      movel([0.226633, -1.444868, -2.521019, -0.746502, 1.570796, 1.797429],accel_mss,speed_ms,0,blend_radius_m)
      movel([0.225647, -1.445273, -2.520694, -0.746422, 1.570796, 1.796443],accel_mss,speed_ms,0,blend_radius_m)
      movel([0.224501, -1.445732, -2.520325, -0.746331, 1.570796, 1.795298],accel_mss,speed_ms,0,blend_radius_m)
      movel([0.221549, -1.446906, -2.519382, -0.746101, 1.570796, 1.792346],accel_mss,speed_ms,0,blend_radius_m)
      movel([0.221114, -1.448639, -2.517985, -0.745765, 1.570796, 1.791910],accel_mss,speed_ms,0,blend_radius_m)
      movel([0.220680, -1.450369, -2.516586, -0.745434, 1.570796, 1.791476],accel_mss,speed_ms,0,blend_radius_m)
      movel([0.218279, -1.451481, -2.515684, -0.745224, 1.570796, 1.789076],accel_mss,speed_ms,0,blend_radius_m)
      movel([0.215883, -1.452595, -2.514779, -0.745015, 1.570796, 1.786679],accel_mss,speed_ms,0,blend_radius_m)
      movel([0.215624, -1.453437, -2.514093, -0.744859, 1.570796, 1.786421],accel_mss,speed_ms,0,blend_radius_m)
      movel([0.215367, -1.454275, -2.513410, -0.744704, 1.570796, 1.786163],accel_mss,speed_ms,0,blend_radius_m)
      movel([0.192396, -1.457892, -2.510448, -0.744049, 1.570796, 1.763193],accel_mss,speed_ms,0,blend_radius_m)
      movel([0.169430, -1.461921, -2.507125, -0.743343, 1.570796, 1.740226],accel_mss,speed_ms,0,blend_radius_m)
      movel([0.170007, -1.461323, -2.507620, -0.743446, 1.570796, 1.740803],accel_mss,speed_ms,0,blend_radius_m)
      movel([0.170664, -1.460630, -2.508192, -0.743566, 1.570796, 1.741460],accel_mss,speed_ms,0,blend_radius_m)
      movel([0.171304, -1.459927, -2.508773, -0.743689, 1.570796, 1.742101],accel_mss,speed_ms,0,blend_radius_m)
      movel([0.171930, -1.459214, -2.509360, -0.743814, 1.570796, 1.742727],accel_mss,speed_ms,0,blend_radius_m)
      movel([0.172537, -1.458492, -2.509955, -0.743942, 1.570796, 1.743334],accel_mss,speed_ms,0,blend_radius_m)
      movel([0.173093, -1.457802, -2.510522, -0.744065, 1.570796, 1.743889],accel_mss,speed_ms,0,blend_radius_m)
      movel([0.173629, -1.457105, -2.511094, -0.744190, 1.570796, 1.744425],accel_mss,speed_ms,0,blend_radius_m)
      movel([0.174144, -1.456397, -2.511674, -0.744317, 1.570796, 1.744940],accel_mss,speed_ms,0,blend_radius_m)
      movel([0.174639, -1.455683, -2.512259, -0.744447, 1.570796, 1.745435],accel_mss,speed_ms,0,blend_radius_m)
      movel([0.175094, -1.454986, -2.512830, -0.744574, 1.570796, 1.745891],accel_mss,speed_ms,0,blend_radius_m)
      movel([0.175530, -1.454281, -2.513405, -0.744703, 1.570796, 1.746326],accel_mss,speed_ms,0,blend_radius_m)
      movel([0.175941, -1.453573, -2.513982, -0.744834, 1.570796, 1.746737],accel_mss,speed_ms,0,blend_radius_m)
      movel([0.176327, -1.452859, -2.514564, -0.744966, 1.570796, 1.747124],accel_mss,speed_ms,0,blend_radius_m)
      movel([0.176693, -1.452141, -2.515148, -0.745100, 1.570796, 1.747489],accel_mss,speed_ms,0,blend_radius_m)
      movel([0.177031, -1.451421, -2.515732, -0.745235, 1.570796, 1.747828],accel_mss,speed_ms,0,blend_radius_m)
      movel([0.177346, -1.450701, -2.516317, -0.745371, 1.570796, 1.748142],accel_mss,speed_ms,0,blend_radius_m)
      movel([0.177636, -1.449977, -2.516903, -0.745509, 1.570796, 1.748432],accel_mss,speed_ms,0,blend_radius_m)
      movel([0.177833, -1.449428, -2.517348, -0.745614, 1.570796, 1.748629],accel_mss,speed_ms,0,blend_radius_m)
      movel([0.178004, -1.448880, -2.517790, -0.745719, 1.570796, 1.748800],accel_mss,speed_ms,0,blend_radius_m)
      movel([0.178150, -1.448335, -2.518230, -0.745824, 1.570796, 1.748947],accel_mss,speed_ms,0,blend_radius_m)
      movel([0.178390, -1.447290, -2.519073, -0.746026, 1.570796, 1.749187],accel_mss,speed_ms,0,blend_radius_m)
      movel([0.178595, -1.446248, -2.519911, -0.746230, 1.570796, 1.749391],accel_mss,speed_ms,0,blend_radius_m)
      movel([0.178762, -1.445209, -2.520745, -0.746435, 1.570796, 1.749558],accel_mss,speed_ms,0,blend_radius_m)
      movel([0.178895, -1.444175, -2.521574, -0.746640, 1.570796, 1.749691],accel_mss,speed_ms,0,blend_radius_m)
      movel([0.178940, -1.443633, -2.522007, -0.746748, 1.570796, 1.749736],accel_mss,speed_ms,0,blend_radius_m)
      movel([0.178961, -1.443099, -2.522434, -0.746855, 1.570796, 1.749758],accel_mss,speed_ms,0,blend_radius_m)
      movel([0.178957, -1.442574, -2.522854, -0.746961, 1.570796, 1.749753],accel_mss,speed_ms,0,blend_radius_m)
      movel([0.178923, -1.441954, -2.523348, -0.747086, 1.570796, 1.749719],accel_mss,speed_ms,0,blend_radius_m)
      movel([0.178865, -1.441344, -2.523834, -0.747210, 1.570796, 1.749661],accel_mss,speed_ms,0,blend_radius_m)
      movel([0.178785, -1.440744, -2.524312, -0.747333, 1.570796, 1.749581],accel_mss,speed_ms,0,blend_radius_m)
      movel([0.178683, -1.440151, -2.524784, -0.747455, 1.570796, 1.749480],accel_mss,speed_ms,0,blend_radius_m)
      movel([0.178556, -1.439564, -2.525250, -0.747575, 1.570796, 1.749352],accel_mss,speed_ms,0,blend_radius_m)
      movel([0.178406, -1.438989, -2.525706, -0.747694, 1.570796, 1.749202],accel_mss,speed_ms,0,blend_radius_m)
      movel([0.178233, -1.438423, -2.526154, -0.747812, 1.570796, 1.749030],accel_mss,speed_ms,0,blend_radius_m)
      movel([0.178039, -1.437870, -2.526592, -0.747927, 1.570796, 1.748835],accel_mss,speed_ms,0,blend_radius_m)
      movel([0.177832, -1.437349, -2.527004, -0.748036, 1.570796, 1.748629],accel_mss,speed_ms,0,blend_radius_m)
      movel([0.177600, -1.436843, -2.527404, -0.748143, 1.570796, 1.748397],accel_mss,speed_ms,0,blend_radius_m)
      movel([0.177348, -1.436348, -2.527794, -0.748247, 1.570796, 1.748144],accel_mss,speed_ms,0,blend_radius_m)
      movel([0.177075, -1.435868, -2.528172, -0.748348, 1.570796, 1.747871],accel_mss,speed_ms,0,blend_radius_m)
      movel([0.176803, -1.435445, -2.528506, -0.748438, 1.570796, 1.747599],accel_mss,speed_ms,0,blend_radius_m)
      movel([0.176507, -1.435040, -2.528824, -0.748524, 1.570796, 1.747303],accel_mss,speed_ms,0,blend_radius_m)
      movel([0.176184, -1.434656, -2.529126, -0.748607, 1.570796, 1.746980],accel_mss,speed_ms,0,blend_radius_m)
      movel([0.175838, -1.434288, -2.529416, -0.748685, 1.570796, 1.746634],accel_mss,speed_ms,0,blend_radius_m)
      movel([0.175621, -1.434068, -2.529588, -0.748732, 1.570796, 1.746418],accel_mss,speed_ms,0,blend_radius_m)
      movel([0.175406, -1.433844, -2.529764, -0.748781, 1.570796, 1.746202],accel_mss,speed_ms,0,blend_radius_m)
      movel([0.175223, -1.433647, -2.529919, -0.748823, 1.570796, 1.746019],accel_mss,speed_ms,0,blend_radius_m)
      movel([0.175114, -1.433520, -2.530018, -0.748850, 1.570796, 1.745911],accel_mss,speed_ms,0,blend_radius_m)
      movel([0.175101, -1.433486, -2.530046, -0.748858, 1.570796, 1.745898],accel_mss,speed_ms,0,blend_radius_m)
      movel([0.175103, -1.433444, -2.530078, -0.748867, 1.570796, 1.745899],accel_mss,speed_ms,0,blend_radius_m)
      movel([0.175125, -1.433400, -2.530112, -0.748876, 1.570796, 1.745921],accel_mss,speed_ms,0,blend_radius_m)
      movel([0.175160, -1.433360, -2.530144, -0.748885, 1.570796, 1.745956],accel_mss,speed_ms,0,blend_radius_m)
      movel([0.175206, -1.433328, -2.530169, -0.748892, 1.570796, 1.746003],accel_mss,speed_ms,0,blend_radius_m)
      movel([0.175257, -1.433310, -2.530183, -0.748896, 1.570796, 1.746053],accel_mss,speed_ms,0,blend_radius_m)
      movel([0.176819, -1.432981, -2.530441, -0.748967, 1.570796, 1.747615],accel_mss,speed_ms,0,blend_radius_m)
      movel([0.178381, -1.432663, -2.530691, -0.749036, 1.570796, 1.749177],accel_mss,speed_ms,0,blend_radius_m)
      movel([0.181096, -1.432128, -2.531109, -0.749152, 1.570796, 1.751892],accel_mss,speed_ms,0,blend_radius_m)
      movel([0.183811, -1.431613, -2.531512, -0.749264, 1.570796, 1.754607],accel_mss,speed_ms,0,blend_radius_m)
      movel([0.198869, -1.428910, -2.533619, -0.749860, 1.570796, 1.769665],accel_mss,speed_ms,0,blend_radius_m)
      movel([0.222820, -1.424984, -2.536660, -0.750745, 1.570796, 1.793616],accel_mss,speed_ms,0,blend_radius_m)
      movel([0.222594, -1.426095, -2.535802, -0.750492, 1.570796, 1.793390],accel_mss,speed_ms,0,blend_radius_m)
      movel([0.222367, -1.427201, -2.534946, -0.750242, 1.570796, 1.793163],accel_mss,speed_ms,0,blend_radius_m)
      movel([0.224300, -1.427644, -2.534602, -0.750143, 1.570796, 1.795096],accel_mss,speed_ms,0,blend_radius_m)
      movel([0.226229, -1.428093, -2.534254, -0.750042, 1.570796, 1.797025],accel_mss,speed_ms,0,blend_radius_m)
      movel([0.225880, -1.429660, -2.533035, -0.749693, 1.570796, 1.796676],accel_mss,speed_ms,0,blend_radius_m)
      movel([0.225532, -1.431226, -2.531814, -0.749349, 1.570796, 1.796328],accel_mss,speed_ms,0,blend_radius_m)
      movel([0.227778, -1.431582, -2.531536, -0.749271, 1.570796, 1.798574],accel_mss,speed_ms,0,blend_radius_m)
      movel([0.228675, -1.431729, -2.531421, -0.749239, 1.570796, 1.799471],accel_mss,speed_ms,0,blend_radius_m)
      movel([0.229514, -1.431876, -2.531306, -0.749207, 1.570796, 1.800311],accel_mss,speed_ms,0,blend_radius_m)
      movel([0.230217, -1.432003, -2.531207, -0.749179, 1.570796, 1.801013],accel_mss,speed_ms,0,blend_radius_m)
      movel([0.230379, -1.432035, -2.531182, -0.749172, 1.570796, 1.801175],accel_mss,speed_ms,0,blend_radius_m)
      movel([0.230535, -1.432072, -2.531153, -0.749164, 1.570796, 1.801331],accel_mss,speed_ms,0,blend_radius_m)
      movel([0.231052, -1.432199, -2.531054, -0.749136, 1.570796, 1.801848],accel_mss,speed_ms,0,blend_radius_m)
      speed_ms = 0.003
      movel([0.231052, -1.435336, -2.532457, -0.744595, 1.570796, 1.801848],accel_mss,speed_ms,0,blend_radius_m)
      speed_ms = 0.007
      movel([0.229385, -1.441407, -2.527656, -0.743326, 1.570796, 1.800181],accel_mss,speed_ms,0,blend_radius_m)
      movel([0.228744, -1.443727, -2.525806, -0.742856, 1.570796, 1.799541],accel_mss,speed_ms,0,blend_radius_m)
      movel([0.228465, -1.444712, -2.525018, -0.742659, 1.570796, 1.799261],accel_mss,speed_ms,0,blend_radius_m)
      movel([0.228181, -1.445697, -2.524229, -0.742463, 1.570796, 1.798977],accel_mss,speed_ms,0,blend_radius_m)
      movel([0.227676, -1.447436, -2.522832, -0.742122, 1.570796, 1.798473],accel_mss,speed_ms,0,blend_radius_m)
      movel([0.227660, -1.447473, -2.522802, -0.742114, 1.570796, 1.798457],accel_mss,speed_ms,0,blend_radius_m)
      movel([0.227635, -1.447510, -2.522772, -0.742107, 1.570796, 1.798432],accel_mss,speed_ms,0,blend_radius_m)
      movel([0.227601, -1.447542, -2.522746, -0.742101, 1.570796, 1.798397],accel_mss,speed_ms,0,blend_radius_m)
      movel([0.227545, -1.447583, -2.522713, -0.742093, 1.570796, 1.798341],accel_mss,speed_ms,0,blend_radius_m)
      movel([0.227485, -1.447613, -2.522689, -0.742087, 1.570796, 1.798281],accel_mss,speed_ms,0,blend_radius_m)
      movel([0.226633, -1.447968, -2.522403, -0.742018, 1.570796, 1.797429],accel_mss,speed_ms,0,blend_radius_m)
      movel([0.225647, -1.448372, -2.522078, -0.741939, 1.570796, 1.796443],accel_mss,speed_ms,0,blend_radius_m)
      movel([0.224501, -1.448830, -2.521708, -0.741851, 1.570796, 1.795298],accel_mss,speed_ms,0,blend_radius_m)
      movel([0.221549, -1.450000, -2.520763, -0.741626, 1.570796, 1.792346],accel_mss,speed_ms,0,blend_radius_m)
      movel([0.221114, -1.451729, -2.519363, -0.741298, 1.570796, 1.791910],accel_mss,speed_ms,0,blend_radius_m)
      movel([0.220680, -1.453453, -2.517961, -0.740975, 1.570796, 1.791476],accel_mss,speed_ms,0,blend_radius_m)
      movel([0.218279, -1.454562, -2.517058, -0.740769, 1.570796, 1.789076],accel_mss,speed_ms,0,blend_radius_m)
      movel([0.215883, -1.455673, -2.516151, -0.740566, 1.570796, 1.786679],accel_mss,speed_ms,0,blend_radius_m)
      movel([0.215624, -1.456512, -2.515464, -0.740413, 1.570796, 1.786421],accel_mss,speed_ms,0,blend_radius_m)
      movel([0.215367, -1.457348, -2.514779, -0.740262, 1.570796, 1.786163],accel_mss,speed_ms,0,blend_radius_m)
      movel([0.192396, -1.460954, -2.511812, -0.739623, 1.570796, 1.763193],accel_mss,speed_ms,0,blend_radius_m)
      movel([0.169430, -1.464971, -2.508483, -0.738935, 1.570796, 1.740226],accel_mss,speed_ms,0,blend_radius_m)
      movel([0.170007, -1.464375, -2.508979, -0.739036, 1.570796, 1.740803],accel_mss,speed_ms,0,blend_radius_m)
      movel([0.170664, -1.463684, -2.509552, -0.739153, 1.570796, 1.741460],accel_mss,speed_ms,0,blend_radius_m)
      movel([0.171304, -1.462983, -2.510134, -0.739272, 1.570796, 1.742101],accel_mss,speed_ms,0,blend_radius_m)
      movel([0.171930, -1.462273, -2.510722, -0.739394, 1.570796, 1.742727],accel_mss,speed_ms,0,blend_radius_m)
      movel([0.172537, -1.461552, -2.511318, -0.739519, 1.570796, 1.743334],accel_mss,speed_ms,0,blend_radius_m)
      movel([0.173093, -1.460865, -2.511885, -0.739639, 1.570796, 1.743889],accel_mss,speed_ms,0,blend_radius_m)
      movel([0.173629, -1.460169, -2.512459, -0.739760, 1.570796, 1.744425],accel_mss,speed_ms,0,blend_radius_m)
      movel([0.174144, -1.459464, -2.513040, -0.739885, 1.570796, 1.744940],accel_mss,speed_ms,0,blend_radius_m)
      movel([0.174639, -1.458752, -2.513626, -0.740011, 1.570796, 1.745435],accel_mss,speed_ms,0,blend_radius_m)
      movel([0.175094, -1.458056, -2.514198, -0.740135, 1.570796, 1.745891],accel_mss,speed_ms,0,blend_radius_m)
      movel([0.175530, -1.457354, -2.514774, -0.740261, 1.570796, 1.746326],accel_mss,speed_ms,0,blend_radius_m)
      movel([0.175941, -1.456648, -2.515353, -0.740388, 1.570796, 1.746737],accel_mss,speed_ms,0,blend_radius_m)
      movel([0.176327, -1.455936, -2.515935, -0.740518, 1.570796, 1.747124],accel_mss,speed_ms,0,blend_radius_m)
      movel([0.176693, -1.455220, -2.516521, -0.740648, 1.570796, 1.747489],accel_mss,speed_ms,0,blend_radius_m)
      movel([0.177031, -1.454502, -2.517106, -0.740780, 1.570796, 1.747828],accel_mss,speed_ms,0,blend_radius_m)
      movel([0.177346, -1.453784, -2.517691, -0.740913, 1.570796, 1.748142],accel_mss,speed_ms,0,blend_radius_m)
      movel([0.177636, -1.453063, -2.518279, -0.741047, 1.570796, 1.748432],accel_mss,speed_ms,0,blend_radius_m)
      movel([0.177833, -1.452515, -2.518725, -0.741150, 1.570796, 1.748629],accel_mss,speed_ms,0,blend_radius_m)
      movel([0.178004, -1.451969, -2.519168, -0.741252, 1.570796, 1.748800],accel_mss,speed_ms,0,blend_radius_m)
      movel([0.178150, -1.451425, -2.519609, -0.741355, 1.570796, 1.748947],accel_mss,speed_ms,0,blend_radius_m)
      movel([0.178390, -1.450383, -2.520453, -0.741553, 1.570796, 1.749187],accel_mss,speed_ms,0,blend_radius_m)
      movel([0.178595, -1.449344, -2.521293, -0.741752, 1.570796, 1.749391],accel_mss,speed_ms,0,blend_radius_m)
      movel([0.178762, -1.448308, -2.522129, -0.741952, 1.570796, 1.749558],accel_mss,speed_ms,0,blend_radius_m)
      movel([0.178895, -1.447278, -2.522959, -0.742152, 1.570796, 1.749691],accel_mss,speed_ms,0,blend_radius_m)
      movel([0.178940, -1.446737, -2.523393, -0.742258, 1.570796, 1.749736],accel_mss,speed_ms,0,blend_radius_m)
      movel([0.178961, -1.446205, -2.523821, -0.742363, 1.570796, 1.749758],accel_mss,speed_ms,0,blend_radius_m)
      movel([0.178957, -1.445681, -2.524242, -0.742466, 1.570796, 1.749753],accel_mss,speed_ms,0,blend_radius_m)
      movel([0.178923, -1.445063, -2.524737, -0.742589, 1.570796, 1.749719],accel_mss,speed_ms,0,blend_radius_m)
      movel([0.178865, -1.444455, -2.525224, -0.742710, 1.570796, 1.749661],accel_mss,speed_ms,0,blend_radius_m)
      movel([0.178785, -1.443856, -2.525703, -0.742830, 1.570796, 1.749581],accel_mss,speed_ms,0,blend_radius_m)
      movel([0.178683, -1.443265, -2.526175, -0.742949, 1.570796, 1.749480],accel_mss,speed_ms,0,blend_radius_m)
      movel([0.178556, -1.442680, -2.526642, -0.743067, 1.570796, 1.749352],accel_mss,speed_ms,0,blend_radius_m)
      movel([0.178406, -1.442107, -2.527099, -0.743184, 1.570796, 1.749202],accel_mss,speed_ms,0,blend_radius_m)
      movel([0.178233, -1.441543, -2.527548, -0.743298, 1.570796, 1.749030],accel_mss,speed_ms,0,blend_radius_m)
      movel([0.178039, -1.440990, -2.527987, -0.743411, 1.570796, 1.748835],accel_mss,speed_ms,0,blend_radius_m)
      movel([0.177832, -1.440471, -2.528400, -0.743518, 1.570796, 1.748629],accel_mss,speed_ms,0,blend_radius_m)
      movel([0.177600, -1.439966, -2.528800, -0.743622, 1.570796, 1.748397],accel_mss,speed_ms,0,blend_radius_m)
      movel([0.177348, -1.439473, -2.529192, -0.743724, 1.570796, 1.748144],accel_mss,speed_ms,0,blend_radius_m)
      movel([0.177075, -1.438995, -2.529570, -0.743824, 1.570796, 1.747871],accel_mss,speed_ms,0,blend_radius_m)
      movel([0.176803, -1.438573, -2.529904, -0.743912, 1.570796, 1.747599],accel_mss,speed_ms,0,blend_radius_m)
      movel([0.176507, -1.438169, -2.530224, -0.743996, 1.570796, 1.747303],accel_mss,speed_ms,0,blend_radius_m)
      movel([0.176184, -1.437786, -2.530526, -0.744076, 1.570796, 1.746980],accel_mss,speed_ms,0,blend_radius_m)
      movel([0.175838, -1.437419, -2.530816, -0.744154, 1.570796, 1.746634],accel_mss,speed_ms,0,blend_radius_m)
      movel([0.175621, -1.437200, -2.530989, -0.744200, 1.570796, 1.746418],accel_mss,speed_ms,0,blend_radius_m)
      movel([0.175406, -1.436976, -2.531166, -0.744247, 1.570796, 1.746202],accel_mss,speed_ms,0,blend_radius_m)
      movel([0.175223, -1.436780, -2.531320, -0.744288, 1.570796, 1.746019],accel_mss,speed_ms,0,blend_radius_m)
      movel([0.175114, -1.436654, -2.531420, -0.744315, 1.570796, 1.745911],accel_mss,speed_ms,0,blend_radius_m)
      movel([0.175101, -1.436619, -2.531447, -0.744322, 1.570796, 1.745898],accel_mss,speed_ms,0,blend_radius_m)
      movel([0.175103, -1.436578, -2.531480, -0.744331, 1.570796, 1.745899],accel_mss,speed_ms,0,blend_radius_m)
      movel([0.175125, -1.436534, -2.531514, -0.744340, 1.570796, 1.745921],accel_mss,speed_ms,0,blend_radius_m)
      movel([0.175160, -1.436494, -2.531546, -0.744349, 1.570796, 1.745956],accel_mss,speed_ms,0,blend_radius_m)
      movel([0.175206, -1.436462, -2.531571, -0.744356, 1.570796, 1.746003],accel_mss,speed_ms,0,blend_radius_m)
      movel([0.175257, -1.436444, -2.531585, -0.744359, 1.570796, 1.746053],accel_mss,speed_ms,0,blend_radius_m)
      movel([0.176819, -1.436116, -2.531844, -0.744429, 1.570796, 1.747615],accel_mss,speed_ms,0,blend_radius_m)
      movel([0.178381, -1.435799, -2.532094, -0.744497, 1.570796, 1.749177],accel_mss,speed_ms,0,blend_radius_m)
      movel([0.181096, -1.435266, -2.532513, -0.744610, 1.570796, 1.751892],accel_mss,speed_ms,0,blend_radius_m)
      movel([0.183811, -1.434752, -2.532916, -0.744720, 1.570796, 1.754607],accel_mss,speed_ms,0,blend_radius_m)
      movel([0.198869, -1.432056, -2.535028, -0.745304, 1.570796, 1.769665],accel_mss,speed_ms,0,blend_radius_m)
      movel([0.222820, -1.428142, -2.538075, -0.746172, 1.570796, 1.793616],accel_mss,speed_ms,0,blend_radius_m)
      movel([0.222594, -1.429249, -2.537216, -0.745924, 1.570796, 1.793390],accel_mss,speed_ms,0,blend_radius_m)
      movel([0.222367, -1.430353, -2.536357, -0.745679, 1.570796, 1.793163],accel_mss,speed_ms,0,blend_radius_m)
      movel([0.224300, -1.430794, -2.536013, -0.745581, 1.570796, 1.795096],accel_mss,speed_ms,0,blend_radius_m)
      movel([0.226229, -1.431242, -2.535664, -0.745483, 1.570796, 1.797025],accel_mss,speed_ms,0,blend_radius_m)
      movel([0.225880, -1.432805, -2.534443, -0.745141, 1.570796, 1.796676],accel_mss,speed_ms,0,blend_radius_m)
      movel([0.225532, -1.434366, -2.533220, -0.744803, 1.570796, 1.796328],accel_mss,speed_ms,0,blend_radius_m)
      movel([0.227778, -1.434721, -2.532941, -0.744727, 1.570796, 1.798574],accel_mss,speed_ms,0,blend_radius_m)
      movel([0.228675, -1.434868, -2.532825, -0.744696, 1.570796, 1.799471],accel_mss,speed_ms,0,blend_radius_m)
      movel([0.229514, -1.435014, -2.532711, -0.744664, 1.570796, 1.800311],accel_mss,speed_ms,0,blend_radius_m)
      movel([0.230217, -1.435141, -2.532611, -0.744637, 1.570796, 1.801013],accel_mss,speed_ms,0,blend_radius_m)
      movel([0.230379, -1.435173, -2.532586, -0.744630, 1.570796, 1.801175],accel_mss,speed_ms,0,blend_radius_m)
      movel([0.230535, -1.435210, -2.532557, -0.744622, 1.570796, 1.801331],accel_mss,speed_ms,0,blend_radius_m)
      movel([0.231052, -1.435336, -2.532457, -0.744595, 1.570796, 1.801848],accel_mss,speed_ms,0,blend_radius_m)
      speed_ms = 0.003
      movel([0.231052, -1.422904, -2.526792, -0.762693, 1.570796, 1.801848],accel_mss,speed_ms,0,blend_radius_m)
      speed_ms = 0.01
      movel([0.231052, -1.398971, -2.515069, -0.798349, 1.570796, 1.801848],accel_mss,speed_ms,0,blend_radius_m)
      movel([0.226061, -1.375510, -2.532139, -0.804740, 1.570796, 1.796858],accel_mss,speed_ms,0,blend_radius_m)
      movel([0.226061, -1.399891, -2.544153, -0.768345, 1.570796, 1.796858],accel_mss,speed_ms,0,blend_radius_m)
      speed_ms = 0.003
      movel([0.226061, -1.409374, -2.548523, -0.754492, 1.570796, 1.796858],accel_mss,speed_ms,0,blend_radius_m)
      speed_ms = 0.007
      movel([0.201671, -1.413475, -2.545441, -0.753472, 1.570796, 1.772468],accel_mss,speed_ms,0,blend_radius_m)
      movel([0.177286, -1.418040, -2.541982, -0.752367, 1.570796, 1.748082],accel_mss,speed_ms,0,blend_radius_m)
      movel([0.178865, -1.416483, -2.543165, -0.752740, 1.570796, 1.749661],accel_mss,speed_ms,0,blend_radius_m)
      movel([0.179419, -1.415928, -2.543587, -0.752874, 1.570796, 1.750215],accel_mss,speed_ms,0,blend_radius_m)
      movel([0.179959, -1.415365, -2.544013, -0.753011, 1.570796, 1.750755],accel_mss,speed_ms,0,blend_radius_m)
      movel([0.180490, -1.414793, -2.544446, -0.753150, 1.570796, 1.751286],accel_mss,speed_ms,0,blend_radius_m)
      movel([0.181005, -1.414212, -2.544886, -0.753292, 1.570796, 1.751801],accel_mss,speed_ms,0,blend_radius_m)
      movel([0.181508, -1.413624, -2.545329, -0.753436, 1.570796, 1.752305],accel_mss,speed_ms,0,blend_radius_m)
      movel([0.181997, -1.413031, -2.545776, -0.753581, 1.570796, 1.752794],accel_mss,speed_ms,0,blend_radius_m)
      movel([0.182473, -1.412431, -2.546229, -0.753729, 1.570796, 1.753269],accel_mss,speed_ms,0,blend_radius_m)
      movel([0.182934, -1.411822, -2.546687, -0.753880, 1.570796, 1.753730],accel_mss,speed_ms,0,blend_radius_m)
      movel([0.183381, -1.411210, -2.547147, -0.754032, 1.570796, 1.754177],accel_mss,speed_ms,0,blend_radius_m)
      movel([0.183807, -1.410599, -2.547605, -0.754184, 1.570796, 1.754603],accel_mss,speed_ms,0,blend_radius_m)
      movel([0.184216, -1.409985, -2.548066, -0.754338, 1.570796, 1.755012],accel_mss,speed_ms,0,blend_radius_m)
      movel([0.184611, -1.409365, -2.548530, -0.754494, 1.570796, 1.755407],accel_mss,speed_ms,0,blend_radius_m)
      movel([0.184988, -1.408742, -2.548996, -0.754651, 1.570796, 1.755785],accel_mss,speed_ms,0,blend_radius_m)
      movel([0.185349, -1.408116, -2.549464, -0.754809, 1.570796, 1.756145],accel_mss,speed_ms,0,blend_radius_m)
      movel([0.185692, -1.407486, -2.549933, -0.754969, 1.570796, 1.756488],accel_mss,speed_ms,0,blend_radius_m)
      movel([0.186015, -1.406854, -2.550405, -0.755130, 1.570796, 1.756812],accel_mss,speed_ms,0,blend_radius_m)
      movel([0.186323, -1.406222, -2.550875, -0.755292, 1.570796, 1.757119],accel_mss,speed_ms,0,blend_radius_m)
      movel([0.186613, -1.405587, -2.551347, -0.755455, 1.570796, 1.757409],accel_mss,speed_ms,0,blend_radius_m)
      movel([0.186886, -1.404946, -2.551823, -0.755620, 1.570796, 1.757683],accel_mss,speed_ms,0,blend_radius_m)
      movel([0.187141, -1.404306, -2.552297, -0.755786, 1.570796, 1.757938],accel_mss,speed_ms,0,blend_radius_m)
      movel([0.187376, -1.403666, -2.552771, -0.755952, 1.570796, 1.758173],accel_mss,speed_ms,0,blend_radius_m)
      movel([0.187592, -1.403029, -2.553242, -0.756118, 1.570796, 1.758388],accel_mss,speed_ms,0,blend_radius_m)
      movel([0.187790, -1.402390, -2.553714, -0.756285, 1.570796, 1.758586],accel_mss,speed_ms,0,blend_radius_m)
      movel([0.187966, -1.401755, -2.554183, -0.756451, 1.570796, 1.758763],accel_mss,speed_ms,0,blend_radius_m)
      movel([0.188125, -1.401121, -2.554650, -0.756618, 1.570796, 1.758921],accel_mss,speed_ms,0,blend_radius_m)
      movel([0.188261, -1.400493, -2.555112, -0.756784, 1.570796, 1.759057],accel_mss,speed_ms,0,blend_radius_m)
      movel([0.188378, -1.399865, -2.555573, -0.756951, 1.570796, 1.759175],accel_mss,speed_ms,0,blend_radius_m)
      movel([0.188480, -1.399226, -2.556042, -0.757121, 1.570796, 1.759276],accel_mss,speed_ms,0,blend_radius_m)
      movel([0.188560, -1.398593, -2.556506, -0.757290, 1.570796, 1.759356],accel_mss,speed_ms,0,blend_radius_m)
      movel([0.188622, -1.397964, -2.556966, -0.757458, 1.570796, 1.759418],accel_mss,speed_ms,0,blend_radius_m)
      movel([0.188665, -1.397341, -2.557422, -0.757626, 1.570796, 1.759461],accel_mss,speed_ms,0,blend_radius_m)
      movel([0.188685, -1.396724, -2.557873, -0.757792, 1.570796, 1.759482],accel_mss,speed_ms,0,blend_radius_m)
      movel([0.188688, -1.396112, -2.558319, -0.757958, 1.570796, 1.759485],accel_mss,speed_ms,0,blend_radius_m)
      movel([0.188671, -1.395507, -2.558760, -0.758122, 1.570796, 1.759468],accel_mss,speed_ms,0,blend_radius_m)
      movel([0.188634, -1.394910, -2.559194, -0.758285, 1.570796, 1.759430],accel_mss,speed_ms,0,blend_radius_m)
      movel([0.188579, -1.394318, -2.559624, -0.758446, 1.570796, 1.759375],accel_mss,speed_ms,0,blend_radius_m)
      movel([0.188504, -1.393790, -2.560008, -0.758591, 1.570796, 1.759300],accel_mss,speed_ms,0,blend_radius_m)
      movel([0.188404, -1.393275, -2.560381, -0.758733, 1.570796, 1.759200],accel_mss,speed_ms,0,blend_radius_m)
      movel([0.188276, -1.392773, -2.560745, -0.758871, 1.570796, 1.759072],accel_mss,speed_ms,0,blend_radius_m)
      movel([0.187996, -1.391868, -2.561400, -0.759121, 1.570796, 1.758792],accel_mss,speed_ms,0,blend_radius_m)
      movel([0.187678, -1.390981, -2.562040, -0.759368, 1.570796, 1.758475],accel_mss,speed_ms,0,blend_radius_m)
      movel([0.187325, -1.390131, -2.562653, -0.759605, 1.570796, 1.758121],accel_mss,speed_ms,0,blend_radius_m)
      movel([0.186930, -1.389304, -2.563248, -0.759837, 1.570796, 1.757726],accel_mss,speed_ms,0,blend_radius_m)
      movel([0.186704, -1.388889, -2.563546, -0.759954, 1.570796, 1.757500],accel_mss,speed_ms,0,blend_radius_m)
      movel([0.186451, -1.388494, -2.563830, -0.760065, 1.570796, 1.757247],accel_mss,speed_ms,0,blend_radius_m)
      movel([0.186169, -1.388119, -2.564099, -0.760171, 1.570796, 1.756966],accel_mss,speed_ms,0,blend_radius_m)
      movel([0.185356, -1.387110, -2.564822, -0.760457, 1.570796, 1.756152],accel_mss,speed_ms,0,blend_radius_m)
      movel([0.187278, -1.386614, -2.565177, -0.760598, 1.570796, 1.758074],accel_mss,speed_ms,0,blend_radius_m)
      movel([0.187745, -1.386497, -2.565261, -0.760632, 1.570796, 1.758542],accel_mss,speed_ms,0,blend_radius_m)
      movel([0.188213, -1.386387, -2.565339, -0.760663, 1.570796, 1.759010],accel_mss,speed_ms,0,blend_radius_m)
      movel([0.188677, -1.386287, -2.565410, -0.760691, 1.570796, 1.759474],accel_mss,speed_ms,0,blend_radius_m)
      movel([0.195268, -1.384939, -2.566373, -0.761077, 1.570796, 1.766064],accel_mss,speed_ms,0,blend_radius_m)
      movel([0.199128, -1.384169, -2.566921, -0.761299, 1.570796, 1.769925],accel_mss,speed_ms,0,blend_radius_m)
      movel([0.202988, -1.383416, -2.567457, -0.761517, 1.570796, 1.773784],accel_mss,speed_ms,0,blend_radius_m)
      movel([0.211781, -1.381756, -2.568634, -0.761999, 1.570796, 1.782578],accel_mss,speed_ms,0,blend_radius_m)
      movel([0.234367, -1.377788, -2.571432, -0.763168, 1.570796, 1.805164],accel_mss,speed_ms,0,blend_radius_m)
      movel([0.234061, -1.378967, -2.570604, -0.762819, 1.570796, 1.804857],accel_mss,speed_ms,0,blend_radius_m)
      movel([0.233756, -1.380140, -2.569776, -0.762472, 1.570796, 1.804552],accel_mss,speed_ms,0,blend_radius_m)
      movel([0.234500, -1.380335, -2.569639, -0.762415, 1.570796, 1.805296],accel_mss,speed_ms,0,blend_radius_m)
      movel([0.237966, -1.381179, -2.569042, -0.762168, 1.570796, 1.808763],accel_mss,speed_ms,0,blend_radius_m)
      movel([0.237526, -1.382845, -2.567862, -0.761682, 1.570796, 1.808323],accel_mss,speed_ms,0,blend_radius_m)
      movel([0.237088, -1.384507, -2.566681, -0.761202, 1.570796, 1.807884],accel_mss,speed_ms,0,blend_radius_m)
      movel([0.239898, -1.384948, -2.566366, -0.761075, 1.570796, 1.810695],accel_mss,speed_ms,0,blend_radius_m)
      movel([0.240984, -1.385125, -2.566240, -0.761024, 1.570796, 1.811780],accel_mss,speed_ms,0,blend_radius_m)
      movel([0.241923, -1.385286, -2.566126, -0.760978, 1.570796, 1.812719],accel_mss,speed_ms,0,blend_radius_m)
      movel([0.242731, -1.385428, -2.566024, -0.760937, 1.570796, 1.813528],accel_mss,speed_ms,0,blend_radius_m)
      movel([0.242794, -1.385444, -2.566012, -0.760932, 1.570796, 1.813591],accel_mss,speed_ms,0,blend_radius_m)
      movel([0.242851, -1.385465, -2.565997, -0.760926, 1.570796, 1.813648],accel_mss,speed_ms,0,blend_radius_m)
      movel([0.242882, -1.385488, -2.565981, -0.760920, 1.570796, 1.813679],accel_mss,speed_ms,0,blend_radius_m)
      movel([0.242897, -1.385520, -2.565958, -0.760911, 1.570796, 1.813693],accel_mss,speed_ms,0,blend_radius_m)
      movel([0.242892, -1.385563, -2.565927, -0.760898, 1.570796, 1.813689],accel_mss,speed_ms,0,blend_radius_m)
      movel([0.242698, -1.386351, -2.565365, -0.760673, 1.570796, 1.813495],accel_mss,speed_ms,0,blend_radius_m)
      movel([0.242574, -1.386828, -2.565024, -0.760537, 1.570796, 1.813371],accel_mss,speed_ms,0,blend_radius_m)
      movel([0.242438, -1.387308, -2.564680, -0.760401, 1.570796, 1.813234],accel_mss,speed_ms,0,blend_radius_m)
      movel([0.242267, -1.387893, -2.564261, -0.760235, 1.570796, 1.813063],accel_mss,speed_ms,0,blend_radius_m)
      movel([0.242086, -1.388479, -2.563841, -0.760069, 1.570796, 1.812882],accel_mss,speed_ms,0,blend_radius_m)
      movel([0.241667, -1.389863, -2.562845, -0.759680, 1.570796, 1.812463],accel_mss,speed_ms,0,blend_radius_m)
      movel([0.239242, -1.398639, -2.556473, -0.757278, 1.570796, 1.810038],accel_mss,speed_ms,0,blend_radius_m)
      movel([0.235946, -1.400028, -2.555454, -0.756908, 1.570796, 1.806742],accel_mss,speed_ms,0,blend_radius_m)
      movel([0.232656, -1.401421, -2.554429, -0.756539, 1.570796, 1.803453],accel_mss,speed_ms,0,blend_radius_m)
      movel([0.232176, -1.403269, -2.553065, -0.756055, 1.570796, 1.802972],accel_mss,speed_ms,0,blend_radius_m)
      movel([0.231697, -1.405111, -2.551700, -0.755578, 1.570796, 1.802493],accel_mss,speed_ms,0,blend_radius_m)
      movel([0.229109, -1.406327, -2.550797, -0.755265, 1.570796, 1.799906],accel_mss,speed_ms,0,blend_radius_m)
      movel([0.226526, -1.407545, -2.549889, -0.754954, 1.570796, 1.797322],accel_mss,speed_ms,0,blend_radius_m)
      movel([0.226293, -1.408460, -2.549206, -0.754722, 1.570796, 1.797090],accel_mss,speed_ms,0,blend_radius_m)
      movel([0.226061, -1.409374, -2.548523, -0.754492, 1.570796, 1.796858],accel_mss,speed_ms,0,blend_radius_m)
      speed_ms = 0.003
      movel([0.226061, -1.412577, -2.549963, -0.749849, 1.570796, 1.796858],accel_mss,speed_ms,0,blend_radius_m)
      speed_ms = 0.007
      movel([0.201671, -1.416666, -2.546875, -0.748848, 1.570796, 1.772468],accel_mss,speed_ms,0,blend_radius_m)
      movel([0.177286, -1.421218, -2.543409, -0.747763, 1.570796, 1.748082],accel_mss,speed_ms,0,blend_radius_m)
      movel([0.178865, -1.419666, -2.544594, -0.748129, 1.570796, 1.749661],accel_mss,speed_ms,0,blend_radius_m)
      movel([0.179419, -1.419112, -2.545016, -0.748261, 1.570796, 1.750215],accel_mss,speed_ms,0,blend_radius_m)
      movel([0.179959, -1.418550, -2.545444, -0.748395, 1.570796, 1.750755],accel_mss,speed_ms,0,blend_radius_m)
      movel([0.180490, -1.417980, -2.545878, -0.748531, 1.570796, 1.751286],accel_mss,speed_ms,0,blend_radius_m)
      movel([0.181005, -1.417400, -2.546318, -0.748671, 1.570796, 1.751801],accel_mss,speed_ms,0,blend_radius_m)
      movel([0.181508, -1.416815, -2.546762, -0.748812, 1.570796, 1.752305],accel_mss,speed_ms,0,blend_radius_m)
      movel([0.181997, -1.416224, -2.547210, -0.748955, 1.570796, 1.752794],accel_mss,speed_ms,0,blend_radius_m)
      movel([0.182473, -1.415625, -2.547664, -0.749100, 1.570796, 1.753269],accel_mss,speed_ms,0,blend_radius_m)
      movel([0.182934, -1.415018, -2.548123, -0.749248, 1.570796, 1.753730],accel_mss,speed_ms,0,blend_radius_m)
      movel([0.183381, -1.414407, -2.548584, -0.749398, 1.570796, 1.754177],accel_mss,speed_ms,0,blend_radius_m)
      movel([0.183807, -1.413798, -2.549043, -0.749547, 1.570796, 1.754603],accel_mss,speed_ms,0,blend_radius_m)
      movel([0.184216, -1.413186, -2.549505, -0.749698, 1.570796, 1.755012],accel_mss,speed_ms,0,blend_radius_m)
      movel([0.184611, -1.412568, -2.549970, -0.749851, 1.570796, 1.755407],accel_mss,speed_ms,0,blend_radius_m)
      movel([0.184988, -1.411947, -2.550437, -0.750006, 1.570796, 1.755785],accel_mss,speed_ms,0,blend_radius_m)
      movel([0.185349, -1.411322, -2.550906, -0.750161, 1.570796, 1.756145],accel_mss,speed_ms,0,blend_radius_m)
      movel([0.185692, -1.410694, -2.551376, -0.750318, 1.570796, 1.756488],accel_mss,speed_ms,0,blend_radius_m)
      movel([0.186015, -1.410064, -2.551849, -0.750477, 1.570796, 1.756812],accel_mss,speed_ms,0,blend_radius_m)
      movel([0.186323, -1.409433, -2.552320, -0.750636, 1.570796, 1.757119],accel_mss,speed_ms,0,blend_radius_m)
      movel([0.186613, -1.408800, -2.552793, -0.750796, 1.570796, 1.757409],accel_mss,speed_ms,0,blend_radius_m)
      movel([0.186886, -1.408161, -2.553270, -0.750958, 1.570796, 1.757683],accel_mss,speed_ms,0,blend_radius_m)
      movel([0.187141, -1.407523, -2.553745, -0.751121, 1.570796, 1.757938],accel_mss,speed_ms,0,blend_radius_m)
      movel([0.187376, -1.406884, -2.554220, -0.751284, 1.570796, 1.758173],accel_mss,speed_ms,0,blend_radius_m)
      movel([0.187592, -1.406249, -2.554693, -0.751447, 1.570796, 1.758388],accel_mss,speed_ms,0,blend_radius_m)
      movel([0.187790, -1.405612, -2.555165, -0.751611, 1.570796, 1.758586],accel_mss,speed_ms,0,blend_radius_m)
      movel([0.187966, -1.404979, -2.555635, -0.751775, 1.570796, 1.758763],accel_mss,speed_ms,0,blend_radius_m)
      movel([0.188125, -1.404347, -2.556103, -0.751939, 1.570796, 1.758921],accel_mss,speed_ms,0,blend_radius_m)
      movel([0.188261, -1.403720, -2.556566, -0.752103, 1.570796, 1.759057],accel_mss,speed_ms,0,blend_radius_m)
      movel([0.188378, -1.403095, -2.557028, -0.752266, 1.570796, 1.759175],accel_mss,speed_ms,0,blend_radius_m)
      movel([0.188480, -1.402457, -2.557498, -0.752433, 1.570796, 1.759276],accel_mss,speed_ms,0,blend_radius_m)
      movel([0.188560, -1.401826, -2.557964, -0.752600, 1.570796, 1.759356],accel_mss,speed_ms,0,blend_radius_m)
      movel([0.188622, -1.401199, -2.558425, -0.752765, 1.570796, 1.759418],accel_mss,speed_ms,0,blend_radius_m)
      movel([0.188665, -1.400577, -2.558881, -0.752930, 1.570796, 1.759461],accel_mss,speed_ms,0,blend_radius_m)
      movel([0.188685, -1.399962, -2.559333, -0.753094, 1.570796, 1.759482],accel_mss,speed_ms,0,blend_radius_m)
      movel([0.188688, -1.399351, -2.559781, -0.753257, 1.570796, 1.759485],accel_mss,speed_ms,0,blend_radius_m)
      movel([0.188671, -1.398748, -2.560222, -0.753419, 1.570796, 1.759468],accel_mss,speed_ms,0,blend_radius_m)
      movel([0.188634, -1.398153, -2.560658, -0.753579, 1.570796, 1.759430],accel_mss,speed_ms,0,blend_radius_m)
      movel([0.188579, -1.397563, -2.561089, -0.753738, 1.570796, 1.759375],accel_mss,speed_ms,0,blend_radius_m)
      movel([0.188504, -1.397036, -2.561473, -0.753880, 1.570796, 1.759300],accel_mss,speed_ms,0,blend_radius_m)
      movel([0.188404, -1.396522, -2.561847, -0.754019, 1.570796, 1.759200],accel_mss,speed_ms,0,blend_radius_m)
      movel([0.188276, -1.396022, -2.562211, -0.754155, 1.570796, 1.759072],accel_mss,speed_ms,0,blend_radius_m)
      movel([0.187996, -1.395119, -2.562868, -0.754402, 1.570796, 1.758792],accel_mss,speed_ms,0,blend_radius_m)
      movel([0.187678, -1.394235, -2.563510, -0.754644, 1.570796, 1.758475],accel_mss,speed_ms,0,blend_radius_m)
      movel([0.187325, -1.393387, -2.564124, -0.754878, 1.570796, 1.758121],accel_mss,speed_ms,0,blend_radius_m)
      movel([0.186930, -1.392562, -2.564720, -0.755106, 1.570796, 1.757726],accel_mss,speed_ms,0,blend_radius_m)
      movel([0.186704, -1.392148, -2.565019, -0.755221, 1.570796, 1.757500],accel_mss,speed_ms,0,blend_radius_m)
      movel([0.186451, -1.391754, -2.565304, -0.755331, 1.570796, 1.757247],accel_mss,speed_ms,0,blend_radius_m)
      movel([0.186169, -1.391381, -2.565573, -0.755435, 1.570796, 1.756966],accel_mss,speed_ms,0,blend_radius_m)
      movel([0.185356, -1.390374, -2.566298, -0.755717, 1.570796, 1.756152],accel_mss,speed_ms,0,blend_radius_m)
      movel([0.187278, -1.389880, -2.566654, -0.755856, 1.570796, 1.758074],accel_mss,speed_ms,0,blend_radius_m)
      movel([0.187745, -1.389762, -2.566738, -0.755889, 1.570796, 1.758542],accel_mss,speed_ms,0,blend_radius_m)
      movel([0.188213, -1.389653, -2.566816, -0.755919, 1.570796, 1.759010],accel_mss,speed_ms,0,blend_radius_m)
      movel([0.188677, -1.389554, -2.566888, -0.755947, 1.570796, 1.759474],accel_mss,speed_ms,0,blend_radius_m)
      movel([0.195268, -1.388209, -2.567853, -0.756328, 1.570796, 1.766064],accel_mss,speed_ms,0,blend_radius_m)
      movel([0.199128, -1.387442, -2.568402, -0.756546, 1.570796, 1.769925],accel_mss,speed_ms,0,blend_radius_m)
      movel([0.202988, -1.386690, -2.568939, -0.756760, 1.570796, 1.773784],accel_mss,speed_ms,0,blend_radius_m)
      movel([0.211781, -1.385035, -2.570119, -0.757235, 1.570796, 1.782578],accel_mss,speed_ms,0,blend_radius_m)
      movel([0.234367, -1.381078, -2.572924, -0.758387, 1.570796, 1.805164],accel_mss,speed_ms,0,blend_radius_m)
      movel([0.234061, -1.382253, -2.572093, -0.758043, 1.570796, 1.804857],accel_mss,speed_ms,0,blend_radius_m)
      movel([0.233756, -1.383423, -2.571264, -0.757702, 1.570796, 1.804552],accel_mss,speed_ms,0,blend_radius_m)
      movel([0.234500, -1.383617, -2.571126, -0.757646, 1.570796, 1.805296],accel_mss,speed_ms,0,blend_radius_m)
      movel([0.237966, -1.384460, -2.570528, -0.757401, 1.570796, 1.808763],accel_mss,speed_ms,0,blend_radius_m)
      movel([0.237526, -1.386121, -2.569345, -0.756923, 1.570796, 1.808323],accel_mss,speed_ms,0,blend_radius_m)
      movel([0.237088, -1.387778, -2.568161, -0.756450, 1.570796, 1.807884],accel_mss,speed_ms,0,blend_radius_m)
      movel([0.239898, -1.388219, -2.567845, -0.756325, 1.570796, 1.810695],accel_mss,speed_ms,0,blend_radius_m)
      movel([0.240984, -1.388395, -2.567719, -0.756275, 1.570796, 1.811780],accel_mss,speed_ms,0,blend_radius_m)
      movel([0.241923, -1.388555, -2.567605, -0.756230, 1.570796, 1.812719],accel_mss,speed_ms,0,blend_radius_m)
      movel([0.242731, -1.388697, -2.567502, -0.756189, 1.570796, 1.813528],accel_mss,speed_ms,0,blend_radius_m)
      movel([0.242794, -1.388713, -2.567491, -0.756185, 1.570796, 1.813591],accel_mss,speed_ms,0,blend_radius_m)
      movel([0.242851, -1.388734, -2.567476, -0.756179, 1.570796, 1.813648],accel_mss,speed_ms,0,blend_radius_m)
      movel([0.242882, -1.388757, -2.567460, -0.756172, 1.570796, 1.813679],accel_mss,speed_ms,0,blend_radius_m)
      movel([0.242897, -1.388789, -2.567437, -0.756163, 1.570796, 1.813693],accel_mss,speed_ms,0,blend_radius_m)
      movel([0.242892, -1.388832, -2.567406, -0.756151, 1.570796, 1.813689],accel_mss,speed_ms,0,blend_radius_m)
      movel([0.242698, -1.389618, -2.566842, -0.755929, 1.570796, 1.813495],accel_mss,speed_ms,0,blend_radius_m)
      movel([0.242574, -1.390093, -2.566500, -0.755796, 1.570796, 1.813371],accel_mss,speed_ms,0,blend_radius_m)
      movel([0.242438, -1.390572, -2.566156, -0.755661, 1.570796, 1.813234],accel_mss,speed_ms,0,blend_radius_m)
      movel([0.242267, -1.391155, -2.565736, -0.755498, 1.570796, 1.813063],accel_mss,speed_ms,0,blend_radius_m)
      movel([0.242086, -1.391739, -2.565315, -0.755335, 1.570796, 1.812882],accel_mss,speed_ms,0,blend_radius_m)
      movel([0.241667, -1.393120, -2.564317, -0.754952, 1.570796, 1.812463],accel_mss,speed_ms,0,blend_radius_m)
      movel([0.239242, -1.401871, -2.557930, -0.752588, 1.570796, 1.810038],accel_mss,speed_ms,0,blend_radius_m)
      movel([0.235946, -1.403256, -2.556909, -0.752224, 1.570796, 1.806742],accel_mss,speed_ms,0,blend_radius_m)
      movel([0.232656, -1.404646, -2.555882, -0.751862, 1.570796, 1.803453],accel_mss,speed_ms,0,blend_radius_m)
      movel([0.232176, -1.406488, -2.554515, -0.751386, 1.570796, 1.802972],accel_mss,speed_ms,0,blend_radius_m)
      movel([0.231697, -1.408325, -2.553147, -0.750916, 1.570796, 1.802493],accel_mss,speed_ms,0,blend_radius_m)
      movel([0.229109, -1.409538, -2.552242, -0.750609, 1.570796, 1.799906],accel_mss,speed_ms,0,blend_radius_m)
      movel([0.226526, -1.410753, -2.551332, -0.750304, 1.570796, 1.797322],accel_mss,speed_ms,0,blend_radius_m)
      movel([0.226293, -1.411665, -2.550648, -0.750076, 1.570796, 1.797090],accel_mss,speed_ms,0,blend_radius_m)
      movel([0.226061, -1.412577, -2.549963, -0.749849, 1.570796, 1.796858],accel_mss,speed_ms,0,blend_radius_m)
      speed_ms = 0.003
      movel([0.226061, -1.399891, -2.544153, -0.768345, 1.570796, 1.796858],accel_mss,speed_ms,0,blend_radius_m)
      speed_ms = 0.01
      movel([0.226061, -1.375510, -2.532139, -0.804740, 1.570796, 1.796858],accel_mss,speed_ms,0,blend_radius_m)
      movel([0.183020, -1.374316, -2.532987, -0.805086, 1.570796, 1.753816],accel_mss,speed_ms,0,blend_radius_m)
      movel([0.183020, -1.398719, -2.545016, -0.768653, 1.570796, 1.753816],accel_mss,speed_ms,0,blend_radius_m)
      speed_ms = 0.003
      movel([0.183020, -1.408212, -2.549392, -0.754785, 1.570796, 1.753816],accel_mss,speed_ms,0,blend_radius_m)
      speed_ms = 0.007
      movel([0.182687, -1.408768, -2.548977, -0.754644, 1.570796, 1.753483],accel_mss,speed_ms,0,blend_radius_m)
      movel([0.182341, -1.409322, -2.548562, -0.754505, 1.570796, 1.753138],accel_mss,speed_ms,0,blend_radius_m)
      movel([0.181980, -1.409873, -2.548150, -0.754366, 1.570796, 1.752777],accel_mss,speed_ms,0,blend_radius_m)
      movel([0.181607, -1.410420, -2.547740, -0.754229, 1.570796, 1.752403],accel_mss,speed_ms,0,blend_radius_m)
      movel([0.181221, -1.410962, -2.547333, -0.754094, 1.570796, 1.752017],accel_mss,speed_ms,0,blend_radius_m)
      movel([0.180820, -1.411501, -2.546928, -0.753960, 1.570796, 1.751617],accel_mss,speed_ms,0,blend_radius_m)
      movel([0.180410, -1.412034, -2.546527, -0.753828, 1.570796, 1.751206],accel_mss,speed_ms,0,blend_radius_m)
      movel([0.179994, -1.412549, -2.546140, -0.753700, 1.570796, 1.750790],accel_mss,speed_ms,0,blend_radius_m)
      movel([0.179568, -1.413060, -2.545755, -0.753574, 1.570796, 1.750365],accel_mss,speed_ms,0,blend_radius_m)
      movel([0.179128, -1.413565, -2.545374, -0.753450, 1.570796, 1.749924],accel_mss,speed_ms,0,blend_radius_m)
      movel([0.178681, -1.414064, -2.544997, -0.753328, 1.570796, 1.749477],accel_mss,speed_ms,0,blend_radius_m)
      movel([0.178219, -1.414554, -2.544627, -0.753208, 1.570796, 1.749015],accel_mss,speed_ms,0,blend_radius_m)
      movel([0.177748, -1.415039, -2.544260, -0.753090, 1.570796, 1.748544],accel_mss,speed_ms,0,blend_radius_m)
      movel([0.177267, -1.415515, -2.543900, -0.752975, 1.570796, 1.748064],accel_mss,speed_ms,0,blend_radius_m)
      movel([0.176804, -1.415955, -2.543566, -0.752868, 1.570796, 1.747600],accel_mss,speed_ms,0,blend_radius_m)
      movel([0.176328, -1.416387, -2.543238, -0.752763, 1.570796, 1.747124],accel_mss,speed_ms,0,blend_radius_m)
      movel([0.175846, -1.416811, -2.542917, -0.752661, 1.570796, 1.746642],accel_mss,speed_ms,0,blend_radius_m)
      movel([0.175350, -1.417223, -2.542604, -0.752562, 1.570796, 1.746146],accel_mss,speed_ms,0,blend_radius_m)
      movel([0.174848, -1.417624, -2.542299, -0.752466, 1.570796, 1.745644],accel_mss,speed_ms,0,blend_radius_m)
      movel([0.174337, -1.418015, -2.542001, -0.752373, 1.570796, 1.745133],accel_mss,speed_ms,0,blend_radius_m)
      movel([0.173817, -1.418395, -2.541712, -0.752282, 1.570796, 1.744613],accel_mss,speed_ms,0,blend_radius_m)
      movel([0.173364, -1.418712, -2.541470, -0.752207, 1.570796, 1.744160],accel_mss,speed_ms,0,blend_radius_m)
      movel([0.172906, -1.419024, -2.541232, -0.752133, 1.570796, 1.743702],accel_mss,speed_ms,0,blend_radius_m)
      movel([0.172443, -1.419325, -2.541003, -0.752061, 1.570796, 1.743239],accel_mss,speed_ms,0,blend_radius_m)
      movel([0.171977, -1.419621, -2.540777, -0.751991, 1.570796, 1.742773],accel_mss,speed_ms,0,blend_radius_m)
      movel([0.171509, -1.419904, -2.540560, -0.751924, 1.570796, 1.742306],accel_mss,speed_ms,0,blend_radius_m)
      movel([0.171033, -1.420184, -2.540347, -0.751858, 1.570796, 1.741830],accel_mss,speed_ms,0,blend_radius_m)
      movel([0.170558, -1.420452, -2.540142, -0.751795, 1.570796, 1.741354],accel_mss,speed_ms,0,blend_radius_m)
      movel([0.170077, -1.420712, -2.539942, -0.751734, 1.570796, 1.740873],accel_mss,speed_ms,0,blend_radius_m)
      movel([0.169596, -1.420963, -2.539750, -0.751675, 1.570796, 1.740392],accel_mss,speed_ms,0,blend_radius_m)
      movel([0.169110, -1.421207, -2.539564, -0.751618, 1.570796, 1.739906],accel_mss,speed_ms,0,blend_radius_m)
      movel([0.168636, -1.421433, -2.539391, -0.751565, 1.570796, 1.739433],accel_mss,speed_ms,0,blend_radius_m)
      movel([0.168162, -1.421650, -2.539224, -0.751515, 1.570796, 1.738959],accel_mss,speed_ms,0,blend_radius_m)
      movel([0.167686, -1.421857, -2.539066, -0.751467, 1.570796, 1.738483],accel_mss,speed_ms,0,blend_radius_m)
      movel([0.167210, -1.422055, -2.538914, -0.751420, 1.570796, 1.738006],accel_mss,speed_ms,0,blend_radius_m)
      movel([0.166731, -1.422242, -2.538770, -0.751377, 1.570796, 1.737527],accel_mss,speed_ms,0,blend_radius_m)
      movel([0.166280, -1.422410, -2.538641, -0.751338, 1.570796, 1.737077],accel_mss,speed_ms,0,blend_radius_m)
      movel([0.165830, -1.422565, -2.538522, -0.751302, 1.570796, 1.736627],accel_mss,speed_ms,0,blend_radius_m)
      movel([0.165378, -1.422710, -2.538411, -0.751268, 1.570796, 1.736174],accel_mss,speed_ms,0,blend_radius_m)
      movel([0.164928, -1.422844, -2.538308, -0.751237, 1.570796, 1.735724],accel_mss,speed_ms,0,blend_radius_m)
      movel([0.164480, -1.422965, -2.538215, -0.751209, 1.570796, 1.735276],accel_mss,speed_ms,0,blend_radius_m)
      movel([0.162753, -1.423410, -2.537872, -0.751106, 1.570796, 1.733549],accel_mss,speed_ms,0,blend_radius_m)
      movel([0.163916, -1.416553, -2.543112, -0.752723, 1.570796, 1.734712],accel_mss,speed_ms,0,blend_radius_m)
      movel([0.164210, -1.414839, -2.544411, -0.753139, 1.570796, 1.735007],accel_mss,speed_ms,0,blend_radius_m)
      movel([0.164513, -1.413120, -2.545710, -0.753560, 1.570796, 1.735309],accel_mss,speed_ms,0,blend_radius_m)
      movel([0.165382, -1.408302, -2.549325, -0.754762, 1.570796, 1.736178],accel_mss,speed_ms,0,blend_radius_m)
      movel([0.166353, -1.403026, -2.553245, -0.756119, 1.570796, 1.737149],accel_mss,speed_ms,0,blend_radius_m)
      movel([0.167287, -1.398058, -2.556898, -0.757433, 1.570796, 1.738084],accel_mss,speed_ms,0,blend_radius_m)
      movel([0.169540, -1.386283, -2.565413, -0.760692, 1.570796, 1.740336],accel_mss,speed_ms,0,blend_radius_m)
      movel([0.171435, -1.385975, -2.565634, -0.760780, 1.570796, 1.742231],accel_mss,speed_ms,0,blend_radius_m)
      movel([0.171997, -1.385891, -2.565693, -0.760804, 1.570796, 1.742793],accel_mss,speed_ms,0,blend_radius_m)
      movel([0.172553, -1.385826, -2.565740, -0.760823, 1.570796, 1.743349],accel_mss,speed_ms,0,blend_radius_m)
      movel([0.173104, -1.385776, -2.565775, -0.760837, 1.570796, 1.743900],accel_mss,speed_ms,0,blend_radius_m)
      movel([0.173648, -1.385745, -2.565797, -0.760846, 1.570796, 1.744445],accel_mss,speed_ms,0,blend_radius_m)
      movel([0.174188, -1.385728, -2.565810, -0.760851, 1.570796, 1.744984],accel_mss,speed_ms,0,blend_radius_m)
      movel([0.174719, -1.385730, -2.565808, -0.760850, 1.570796, 1.745515],accel_mss,speed_ms,0,blend_radius_m)
      movel([0.175242, -1.385749, -2.565795, -0.760845, 1.570796, 1.746039],accel_mss,speed_ms,0,blend_radius_m)
      movel([0.175757, -1.385786, -2.565768, -0.760834, 1.570796, 1.746553],accel_mss,speed_ms,0,blend_radius_m)
      movel([0.176261, -1.385839, -2.565731, -0.760819, 1.570796, 1.747057],accel_mss,speed_ms,0,blend_radius_m)
      movel([0.176757, -1.385908, -2.565682, -0.760800, 1.570796, 1.747554],accel_mss,speed_ms,0,blend_radius_m)
      movel([0.177254, -1.385996, -2.565619, -0.760775, 1.570796, 1.748051],accel_mss,speed_ms,0,blend_radius_m)
      movel([0.177741, -1.386099, -2.565545, -0.760745, 1.570796, 1.748537],accel_mss,speed_ms,0,blend_radius_m)
      movel([0.178215, -1.386219, -2.565459, -0.760711, 1.570796, 1.749011],accel_mss,speed_ms,0,blend_radius_m)
      movel([0.178680, -1.386354, -2.565363, -0.760672, 1.570796, 1.749477],accel_mss,speed_ms,0,blend_radius_m)
      movel([0.179133, -1.386507, -2.565253, -0.760629, 1.570796, 1.749929],accel_mss,speed_ms,0,blend_radius_m)
      movel([0.179574, -1.386673, -2.565135, -0.760581, 1.570796, 1.750370],accel_mss,speed_ms,0,blend_radius_m)
      movel([0.180003, -1.386856, -2.565004, -0.760529, 1.570796, 1.750800],accel_mss,speed_ms,0,blend_radius_m)
      movel([0.180418, -1.387053, -2.564863, -0.760473, 1.570796, 1.751214],accel_mss,speed_ms,0,blend_radius_m)
      movel([0.180822, -1.387266, -2.564710, -0.760413, 1.570796, 1.751619],accel_mss,speed_ms,0,blend_radius_m)
      movel([0.181212, -1.387494, -2.564547, -0.760348, 1.570796, 1.752008],accel_mss,speed_ms,0,blend_radius_m)
      movel([0.181597, -1.387741, -2.564370, -0.760278, 1.570796, 1.752393],accel_mss,speed_ms,0,blend_radius_m)
      movel([0.181967, -1.388004, -2.564181, -0.760204, 1.570796, 1.752763],accel_mss,speed_ms,0,blend_radius_m)
      movel([0.182324, -1.388280, -2.563983, -0.760125, 1.570796, 1.753121],accel_mss,speed_ms,0,blend_radius_m)
      movel([0.182665, -1.388570, -2.563775, -0.760044, 1.570796, 1.753461],accel_mss,speed_ms,0,blend_radius_m)
      movel([0.182993, -1.388872, -2.563559, -0.759959, 1.570796, 1.753789],accel_mss,speed_ms,0,blend_radius_m)
      movel([0.183304, -1.389189, -2.563331, -0.759869, 1.570796, 1.754100],accel_mss,speed_ms,0,blend_radius_m)
      movel([0.183600, -1.389519, -2.563093, -0.759777, 1.570796, 1.754396],accel_mss,speed_ms,0,blend_radius_m)
      movel([0.183880, -1.389860, -2.562848, -0.759681, 1.570796, 1.754676],accel_mss,speed_ms,0,blend_radius_m)
      movel([0.184144, -1.390215, -2.562592, -0.759582, 1.570796, 1.754941],accel_mss,speed_ms,0,blend_radius_m)
      movel([0.184393, -1.390581, -2.562329, -0.759480, 1.570796, 1.755189],accel_mss,speed_ms,0,blend_radius_m)
      movel([0.184630, -1.390965, -2.562052, -0.759372, 1.570796, 1.755426],accel_mss,speed_ms,0,blend_radius_m)
      movel([0.184850, -1.391360, -2.561766, -0.759262, 1.570796, 1.755647],accel_mss,speed_ms,0,blend_radius_m)
      movel([0.185057, -1.391767, -2.561472, -0.759149, 1.570796, 1.755853],accel_mss,speed_ms,0,blend_radius_m)
      movel([0.185244, -1.392184, -2.561171, -0.759034, 1.570796, 1.756041],accel_mss,speed_ms,0,blend_radius_m)
      movel([0.185416, -1.392610, -2.560863, -0.758916, 1.570796, 1.756212],accel_mss,speed_ms,0,blend_radius_m)
      movel([0.185574, -1.393045, -2.560548, -0.758796, 1.570796, 1.756370],accel_mss,speed_ms,0,blend_radius_m)
      movel([0.185713, -1.393489, -2.560226, -0.758674, 1.570796, 1.756509],accel_mss,speed_ms,0,blend_radius_m)
      movel([0.185834, -1.393941, -2.559898, -0.758550, 1.570796, 1.756631],accel_mss,speed_ms,0,blend_radius_m)
      movel([0.185941, -1.394404, -2.559562, -0.758423, 1.570796, 1.756738],accel_mss,speed_ms,0,blend_radius_m)
      movel([0.186031, -1.394872, -2.559222, -0.758295, 1.570796, 1.756827],accel_mss,speed_ms,0,blend_radius_m)
      movel([0.186092, -1.395277, -2.558927, -0.758185, 1.570796, 1.756888],accel_mss,speed_ms,0,blend_radius_m)
      movel([0.186138, -1.395687, -2.558628, -0.758073, 1.570796, 1.756934],accel_mss,speed_ms,0,blend_radius_m)
      movel([0.186168, -1.396107, -2.558323, -0.757959, 1.570796, 1.756964],accel_mss,speed_ms,0,blend_radius_m)
      movel([0.186186, -1.396528, -2.558016, -0.757845, 1.570796, 1.756982],accel_mss,speed_ms,0,blend_radius_m)
      movel([0.186186, -1.396957, -2.557703, -0.757729, 1.570796, 1.756982],accel_mss,speed_ms,0,blend_radius_m)
      movel([0.186170, -1.397581, -2.557247, -0.757561, 1.570796, 1.756966],accel_mss,speed_ms,0,blend_radius_m)
      movel([0.186135, -1.398210, -2.556786, -0.757392, 1.570796, 1.756931],accel_mss,speed_ms,0,blend_radius_m)
      movel([0.186082, -1.398845, -2.556322, -0.757222, 1.570796, 1.756878],accel_mss,speed_ms,0,blend_radius_m)
      movel([0.186014, -1.399484, -2.555853, -0.757052, 1.570796, 1.756811],accel_mss,speed_ms,0,blend_radius_m)
      movel([0.185928, -1.400124, -2.555383, -0.756882, 1.570796, 1.756724],accel_mss,speed_ms,0,blend_radius_m)
      movel([0.185822, -1.400769, -2.554909, -0.756711, 1.570796, 1.756619],accel_mss,speed_ms,0,blend_radius_m)
      movel([0.185702, -1.401417, -2.554432, -0.756540, 1.570796, 1.756498],accel_mss,speed_ms,0,blend_radius_m)
      movel([0.185566, -1.402065, -2.553954, -0.756370, 1.570796, 1.756362],accel_mss,speed_ms,0,blend_radius_m)
      movel([0.185458, -1.402513, -2.553623, -0.756253, 1.570796, 1.756254],accel_mss,speed_ms,0,blend_radius_m)
      movel([0.185335, -1.402965, -2.553290, -0.756135, 1.570796, 1.756131],accel_mss,speed_ms,0,blend_radius_m)
      movel([0.185199, -1.403416, -2.552956, -0.756017, 1.570796, 1.755995],accel_mss,speed_ms,0,blend_radius_m)
      movel([0.185049, -1.403868, -2.552621, -0.755899, 1.570796, 1.755845],accel_mss,speed_ms,0,blend_radius_m)
      movel([0.184884, -1.404323, -2.552285, -0.755781, 1.570796, 1.755681],accel_mss,speed_ms,0,blend_radius_m)
      movel([0.184667, -1.404880, -2.551872, -0.755637, 1.570796, 1.755463],accel_mss,speed_ms,0,blend_radius_m)
      movel([0.184430, -1.405438, -2.551458, -0.755493, 1.570796, 1.755227],accel_mss,speed_ms,0,blend_radius_m)
      movel([0.184178, -1.405997, -2.551042, -0.755350, 1.570796, 1.754975],accel_mss,speed_ms,0,blend_radius_m)
      movel([0.183913, -1.406551, -2.550630, -0.755208, 1.570796, 1.754710],accel_mss,speed_ms,0,blend_radius_m)
      movel([0.183630, -1.407107, -2.550216, -0.755066, 1.570796, 1.754426],accel_mss,speed_ms,0,blend_radius_m)
      movel([0.183332, -1.407659, -2.549804, -0.754925, 1.570796, 1.754128],accel_mss,speed_ms,0,blend_radius_m)
      movel([0.183020, -1.408212, -2.549392, -0.754785, 1.570796, 1.753816],accel_mss,speed_ms,0,blend_radius_m)
      speed_ms = 0.003
      movel([0.183020, -1.411417, -2.550834, -0.750137, 1.570796, 1.753816],accel_mss,speed_ms,0,blend_radius_m)
      speed_ms = 0.007
      movel([0.182687, -1.411972, -2.550418, -0.749999, 1.570796, 1.753483],accel_mss,speed_ms,0,blend_radius_m)
      movel([0.182341, -1.412525, -2.550002, -0.749862, 1.570796, 1.753138],accel_mss,speed_ms,0,blend_radius_m)
      movel([0.181980, -1.413074, -2.549589, -0.749726, 1.570796, 1.752777],accel_mss,speed_ms,0,blend_radius_m)
      movel([0.181607, -1.413619, -2.549178, -0.749591, 1.570796, 1.752403],accel_mss,speed_ms,0,blend_radius_m)
      movel([0.181221, -1.414160, -2.548770, -0.749458, 1.570796, 1.752017],accel_mss,speed_ms,0,blend_radius_m)
      movel([0.180820, -1.414698, -2.548365, -0.749327, 1.570796, 1.751617],accel_mss,speed_ms,0,blend_radius_m)
      movel([0.180410, -1.415229, -2.547963, -0.749197, 1.570796, 1.751206],accel_mss,speed_ms,0,blend_radius_m)
      movel([0.179994, -1.415743, -2.547575, -0.749072, 1.570796, 1.750790],accel_mss,speed_ms,0,blend_radius_m)
      movel([0.179568, -1.416252, -2.547189, -0.748948, 1.570796, 1.750365],accel_mss,speed_ms,0,blend_radius_m)
      movel([0.179128, -1.416756, -2.546807, -0.748826, 1.570796, 1.749924],accel_mss,speed_ms,0,blend_radius_m)
      movel([0.178681, -1.417253, -2.546430, -0.748706, 1.570796, 1.749477],accel_mss,speed_ms,0,blend_radius_m)
      movel([0.178219, -1.417742, -2.546058, -0.748589, 1.570796, 1.749015],accel_mss,speed_ms,0,blend_radius_m)
      movel([0.177748, -1.418225, -2.545691, -0.748473, 1.570796, 1.748544],accel_mss,speed_ms,0,blend_radius_m)
      movel([0.177267, -1.418700, -2.545330, -0.748359, 1.570796, 1.748064],accel_mss,speed_ms,0,blend_radius_m)
      movel([0.176804, -1.419139, -2.544996, -0.748255, 1.570796, 1.747600],accel_mss,speed_ms,0,blend_radius_m)
      movel([0.176328, -1.419570, -2.544667, -0.748152, 1.570796, 1.747124],accel_mss,speed_ms,0,blend_radius_m)
      movel([0.175846, -1.419992, -2.544345, -0.748052, 1.570796, 1.746642],accel_mss,speed_ms,0,blend_radius_m)
      movel([0.175350, -1.420403, -2.544031, -0.747955, 1.570796, 1.746146],accel_mss,speed_ms,0,blend_radius_m)
      movel([0.174848, -1.420803, -2.543726, -0.747860, 1.570796, 1.745644],accel_mss,speed_ms,0,blend_radius_m)
      movel([0.174337, -1.421193, -2.543428, -0.747769, 1.570796, 1.745133],accel_mss,speed_ms,0,blend_radius_m)
      movel([0.173817, -1.421572, -2.543137, -0.747680, 1.570796, 1.744613],accel_mss,speed_ms,0,blend_radius_m)
      movel([0.173364, -1.421888, -2.542895, -0.747606, 1.570796, 1.744160],accel_mss,speed_ms,0,blend_radius_m)
      movel([0.172906, -1.422199, -2.542657, -0.747533, 1.570796, 1.743702],accel_mss,speed_ms,0,blend_radius_m)
      movel([0.172443, -1.422499, -2.542427, -0.747463, 1.570796, 1.743239],accel_mss,speed_ms,0,blend_radius_m)
      movel([0.171977, -1.422794, -2.542201, -0.747394, 1.570796, 1.742773],accel_mss,speed_ms,0,blend_radius_m)
      movel([0.171509, -1.423077, -2.541983, -0.747328, 1.570796, 1.742306],accel_mss,speed_ms,0,blend_radius_m)
      movel([0.171033, -1.423356, -2.541769, -0.747264, 1.570796, 1.741830],accel_mss,speed_ms,0,blend_radius_m)
      movel([0.170558, -1.423623, -2.541564, -0.747202, 1.570796, 1.741354],accel_mss,speed_ms,0,blend_radius_m)
      movel([0.170077, -1.423883, -2.541364, -0.747142, 1.570796, 1.740873],accel_mss,speed_ms,0,blend_radius_m)
      movel([0.169596, -1.424133, -2.541172, -0.747084, 1.570796, 1.740392],accel_mss,speed_ms,0,blend_radius_m)
      movel([0.169110, -1.424376, -2.540985, -0.747028, 1.570796, 1.739906],accel_mss,speed_ms,0,blend_radius_m)
      movel([0.168636, -1.424601, -2.540812, -0.746976, 1.570796, 1.739433],accel_mss,speed_ms,0,blend_radius_m)
      movel([0.168162, -1.424818, -2.540645, -0.746927, 1.570796, 1.738959],accel_mss,speed_ms,0,blend_radius_m)
      movel([0.167686, -1.425024, -2.540486, -0.746879, 1.570796, 1.738483],accel_mss,speed_ms,0,blend_radius_m)
      movel([0.167210, -1.425222, -2.540333, -0.746834, 1.570796, 1.738006],accel_mss,speed_ms,0,blend_radius_m)
      movel([0.166731, -1.425408, -2.540189, -0.746791, 1.570796, 1.737527],accel_mss,speed_ms,0,blend_radius_m)
      movel([0.166280, -1.425575, -2.540061, -0.746753, 1.570796, 1.737077],accel_mss,speed_ms,0,blend_radius_m)
      movel([0.165830, -1.425730, -2.539941, -0.746718, 1.570796, 1.736627],accel_mss,speed_ms,0,blend_radius_m)
      movel([0.165378, -1.425874, -2.539830, -0.746685, 1.570796, 1.736174],accel_mss,speed_ms,0,blend_radius_m)
      movel([0.164928, -1.426008, -2.539727, -0.746654, 1.570796, 1.735724],accel_mss,speed_ms,0,blend_radius_m)
      movel([0.164480, -1.426129, -2.539633, -0.746627, 1.570796, 1.735276],accel_mss,speed_ms,0,blend_radius_m)
      movel([0.162753, -1.426573, -2.539290, -0.746526, 1.570796, 1.733549],accel_mss,speed_ms,0,blend_radius_m)
      movel([0.163916, -1.419735, -2.544541, -0.748113, 1.570796, 1.734712],accel_mss,speed_ms,0,blend_radius_m)
      movel([0.164210, -1.418027, -2.545842, -0.748520, 1.570796, 1.735007],accel_mss,speed_ms,0,blend_radius_m)
      movel([0.164513, -1.416312, -2.547144, -0.748934, 1.570796, 1.735309],accel_mss,speed_ms,0,blend_radius_m)
      movel([0.165382, -1.411507, -2.550767, -0.750115, 1.570796, 1.736178],accel_mss,speed_ms,0,blend_radius_m)
      movel([0.166353, -1.406246, -2.554695, -0.751448, 1.570796, 1.737149],accel_mss,speed_ms,0,blend_radius_m)
      movel([0.167287, -1.401292, -2.558356, -0.752741, 1.570796, 1.738084],accel_mss,speed_ms,0,blend_radius_m)
      movel([0.169540, -1.389550, -2.566891, -0.755948, 1.570796, 1.740336],accel_mss,speed_ms,0,blend_radius_m)
      movel([0.171435, -1.389242, -2.567112, -0.756035, 1.570796, 1.742231],accel_mss,speed_ms,0,blend_radius_m)
      movel([0.171997, -1.389159, -2.567172, -0.756059, 1.570796, 1.742793],accel_mss,speed_ms,0,blend_radius_m)
      movel([0.172553, -1.389093, -2.567218, -0.756077, 1.570796, 1.743349],accel_mss,speed_ms,0,blend_radius_m)
      movel([0.173104, -1.389044, -2.567254, -0.756091, 1.570796, 1.743900],accel_mss,speed_ms,0,blend_radius_m)
      movel([0.173648, -1.389013, -2.567276, -0.756100, 1.570796, 1.744445],accel_mss,speed_ms,0,blend_radius_m)
      movel([0.174188, -1.388996, -2.567288, -0.756105, 1.570796, 1.744984],accel_mss,speed_ms,0,blend_radius_m)
      movel([0.174719, -1.388998, -2.567287, -0.756104, 1.570796, 1.745515],accel_mss,speed_ms,0,blend_radius_m)
      movel([0.175242, -1.389017, -2.567273, -0.756099, 1.570796, 1.746039],accel_mss,speed_ms,0,blend_radius_m)
      movel([0.175757, -1.389054, -2.567247, -0.756088, 1.570796, 1.746553],accel_mss,speed_ms,0,blend_radius_m)
      movel([0.176261, -1.389106, -2.567209, -0.756074, 1.570796, 1.747057],accel_mss,speed_ms,0,blend_radius_m)
      movel([0.176757, -1.389175, -2.567160, -0.756054, 1.570796, 1.747554],accel_mss,speed_ms,0,blend_radius_m)
      movel([0.177254, -1.389263, -2.567097, -0.756029, 1.570796, 1.748051],accel_mss,speed_ms,0,blend_radius_m)
      movel([0.177741, -1.389366, -2.567023, -0.756000, 1.570796, 1.748537],accel_mss,speed_ms,0,blend_radius_m)
      movel([0.178215, -1.389486, -2.566937, -0.755967, 1.570796, 1.749011],accel_mss,speed_ms,0,blend_radius_m)
      movel([0.178680, -1.389621, -2.566840, -0.755929, 1.570796, 1.749477],accel_mss,speed_ms,0,blend_radius_m)
      movel([0.179133, -1.389773, -2.566730, -0.755886, 1.570796, 1.749929],accel_mss,speed_ms,0,blend_radius_m)
      movel([0.179574, -1.389938, -2.566612, -0.755839, 1.570796, 1.750370],accel_mss,speed_ms,0,blend_radius_m)
      movel([0.180003, -1.390121, -2.566480, -0.755788, 1.570796, 1.750800],accel_mss,speed_ms,0,blend_radius_m)
      movel([0.180418, -1.390317, -2.566339, -0.755733, 1.570796, 1.751214],accel_mss,speed_ms,0,blend_radius_m)
      movel([0.180822, -1.390530, -2.566186, -0.755673, 1.570796, 1.751619],accel_mss,speed_ms,0,blend_radius_m)
      movel([0.181212, -1.390757, -2.566023, -0.755609, 1.570796, 1.752008],accel_mss,speed_ms,0,blend_radius_m)
      movel([0.181597, -1.391004, -2.565845, -0.755540, 1.570796, 1.752393],accel_mss,speed_ms,0,blend_radius_m)
      movel([0.181967, -1.391266, -2.565656, -0.755467, 1.570796, 1.752763],accel_mss,speed_ms,0,blend_radius_m)
      movel([0.182324, -1.391541, -2.565457, -0.755390, 1.570796, 1.753121],accel_mss,speed_ms,0,blend_radius_m)
      movel([0.182665, -1.391831, -2.565249, -0.755310, 1.570796, 1.753461],accel_mss,speed_ms,0,blend_radius_m)
      movel([0.182993, -1.392131, -2.565032, -0.755226, 1.570796, 1.753789],accel_mss,speed_ms,0,blend_radius_m)
      movel([0.183304, -1.392447, -2.564803, -0.755138, 1.570796, 1.754100],accel_mss,speed_ms,0,blend_radius_m)
      movel([0.183600, -1.392777, -2.564565, -0.755047, 1.570796, 1.754396],accel_mss,speed_ms,0,blend_radius_m)
      movel([0.183880, -1.393116, -2.564320, -0.754953, 1.570796, 1.754676],accel_mss,speed_ms,0,blend_radius_m)
      movel([0.184144, -1.393471, -2.564063, -0.754855, 1.570796, 1.754941],accel_mss,speed_ms,0,blend_radius_m)
      movel([0.184393, -1.393835, -2.563799, -0.754754, 1.570796, 1.755189],accel_mss,speed_ms,0,blend_radius_m)
      movel([0.184630, -1.394218, -2.563522, -0.754649, 1.570796, 1.755426],accel_mss,speed_ms,0,blend_radius_m)
      movel([0.184850, -1.394613, -2.563235, -0.754541, 1.570796, 1.755647],accel_mss,speed_ms,0,blend_radius_m)
      movel([0.185057, -1.395019, -2.562941, -0.754429, 1.570796, 1.755853],accel_mss,speed_ms,0,blend_radius_m)
      movel([0.185244, -1.395434, -2.562639, -0.754316, 1.570796, 1.756041],accel_mss,speed_ms,0,blend_radius_m)
      movel([0.185416, -1.395859, -2.562330, -0.754200, 1.570796, 1.756212],accel_mss,speed_ms,0,blend_radius_m)
      movel([0.185574, -1.396293, -2.562015, -0.754082, 1.570796, 1.756370],accel_mss,speed_ms,0,blend_radius_m)
      movel([0.185713, -1.396736, -2.561692, -0.753961, 1.570796, 1.756509],accel_mss,speed_ms,0,blend_radius_m)
      movel([0.185834, -1.397187, -2.561363, -0.753839, 1.570796, 1.756631],accel_mss,speed_ms,0,blend_radius_m)
      movel([0.185941, -1.397648, -2.561026, -0.753715, 1.570796, 1.756738],accel_mss,speed_ms,0,blend_radius_m)
      movel([0.186031, -1.398115, -2.560685, -0.753589, 1.570796, 1.756827],accel_mss,speed_ms,0,blend_radius_m)
      movel([0.186092, -1.398519, -2.560390, -0.753480, 1.570796, 1.756888],accel_mss,speed_ms,0,blend_radius_m)
      movel([0.186138, -1.398928, -2.560091, -0.753370, 1.570796, 1.756934],accel_mss,speed_ms,0,blend_radius_m)
      movel([0.186168, -1.399346, -2.559784, -0.753258, 1.570796, 1.756964],accel_mss,speed_ms,0,blend_radius_m)
      movel([0.186186, -1.399766, -2.559477, -0.753146, 1.570796, 1.756982],accel_mss,speed_ms,0,blend_radius_m)
      movel([0.186186, -1.400194, -2.559163, -0.753032, 1.570796, 1.756982],accel_mss,speed_ms,0,blend_radius_m)
      movel([0.186170, -1.400816, -2.558706, -0.752867, 1.570796, 1.756966],accel_mss,speed_ms,0,blend_radius_m)
      movel([0.186135, -1.401444, -2.558244, -0.752701, 1.570796, 1.756931],accel_mss,speed_ms,0,blend_radius_m)
      movel([0.186082, -1.402077, -2.557779, -0.752534, 1.570796, 1.756878],accel_mss,speed_ms,0,blend_radius_m)
      movel([0.186014, -1.402714, -2.557309, -0.752366, 1.570796, 1.756811],accel_mss,speed_ms,0,blend_radius_m)
      movel([0.185928, -1.403352, -2.556838, -0.752199, 1.570796, 1.756724],accel_mss,speed_ms,0,blend_radius_m)
      movel([0.185822, -1.403996, -2.556363, -0.752031, 1.570796, 1.756619],accel_mss,speed_ms,0,blend_radius_m)
      movel([0.185702, -1.404641, -2.555885, -0.751863, 1.570796, 1.756498],accel_mss,speed_ms,0,blend_radius_m)
      movel([0.185566, -1.405288, -2.555406, -0.751695, 1.570796, 1.756362],accel_mss,speed_ms,0,blend_radius_m)
      movel([0.185458, -1.405735, -2.555074, -0.751580, 1.570796, 1.756254],accel_mss,speed_ms,0,blend_radius_m)
      movel([0.185335, -1.406185, -2.554740, -0.751464, 1.570796, 1.756131],accel_mss,speed_ms,0,blend_radius_m)
      movel([0.185199, -1.406636, -2.554405, -0.751348, 1.570796, 1.755995],accel_mss,speed_ms,0,blend_radius_m)
      movel([0.185049, -1.407086, -2.554070, -0.751232, 1.570796, 1.755845],accel_mss,speed_ms,0,blend_radius_m)
      movel([0.184884, -1.407540, -2.553733, -0.751117, 1.570796, 1.755681],accel_mss,speed_ms,0,blend_radius_m)
      movel([0.184667, -1.408095, -2.553319, -0.750975, 1.570796, 1.755463],accel_mss,speed_ms,0,blend_radius_m)
      movel([0.184430, -1.408651, -2.552904, -0.750834, 1.570796, 1.755227],accel_mss,speed_ms,0,blend_radius_m)
      movel([0.184178, -1.409209, -2.552488, -0.750692, 1.570796, 1.754975],accel_mss,speed_ms,0,blend_radius_m)
      movel([0.183913, -1.409762, -2.552075, -0.750553, 1.570796, 1.754710],accel_mss,speed_ms,0,blend_radius_m)
      movel([0.183630, -1.410316, -2.551660, -0.750413, 1.570796, 1.754426],accel_mss,speed_ms,0,blend_radius_m)
      movel([0.183332, -1.410867, -2.551247, -0.750275, 1.570796, 1.754128],accel_mss,speed_ms,0,blend_radius_m)
      movel([0.183020, -1.411417, -2.550834, -0.750137, 1.570796, 1.753816],accel_mss,speed_ms,0,blend_radius_m)
      speed_ms = 0.003
      movel([0.183020, -1.398719, -2.545016, -0.768653, 1.570796, 1.753816],accel_mss,speed_ms,0,blend_radius_m)
      speed_ms = 0.01
      movel([0.183020, -1.374316, -2.532987, -0.805086, 1.570796, 1.753816],accel_mss,speed_ms,0,blend_radius_m)
      movel([0.168842, -1.399903, -2.514375, -0.798111, 1.570796, 1.739639],accel_mss,speed_ms,0,blend_radius_m)
      movel([0.168842, -1.423819, -2.526086, -0.762484, 1.570796, 1.739639],accel_mss,speed_ms,0,blend_radius_m)
      speed_ms = 0.003
      movel([0.168842, -1.433106, -2.530343, -0.748940, 1.570796, 1.739639],accel_mss,speed_ms,0,blend_radius_m)
      speed_ms = 0.007
      movel([0.169285, -1.433239, -2.530239, -0.748911, 1.570796, 1.740082],accel_mss,speed_ms,0,blend_radius_m)
      movel([0.169716, -1.433386, -2.530124, -0.748879, 1.570796, 1.740513],accel_mss,speed_ms,0,blend_radius_m)
      movel([0.170138, -1.433545, -2.529999, -0.748845, 1.570796, 1.740935],accel_mss,speed_ms,0,blend_radius_m)
      movel([0.170548, -1.433720, -2.529862, -0.748807, 1.570796, 1.741344],accel_mss,speed_ms,0,blend_radius_m)
      movel([0.170948, -1.433909, -2.529713, -0.748767, 1.570796, 1.741744],accel_mss,speed_ms,0,blend_radius_m)
      movel([0.171334, -1.434111, -2.529555, -0.748723, 1.570796, 1.742130],accel_mss,speed_ms,0,blend_radius_m)
      movel([0.171708, -1.434326, -2.529385, -0.748677, 1.570796, 1.742505],accel_mss,speed_ms,0,blend_radius_m)
      movel([0.172069, -1.434555, -2.529206, -0.748628, 1.570796, 1.742865],accel_mss,speed_ms,0,blend_radius_m)
      movel([0.172417, -1.434795, -2.529017, -0.748577, 1.570796, 1.743214],accel_mss,speed_ms,0,blend_radius_m)
      movel([0.172752, -1.435050, -2.528816, -0.748522, 1.570796, 1.743548],accel_mss,speed_ms,0,blend_radius_m)
      movel([0.173073, -1.435318, -2.528606, -0.748465, 1.570796, 1.743869],accel_mss,speed_ms,0,blend_radius_m)
      movel([0.173380, -1.435596, -2.528387, -0.748406, 1.570796, 1.744176],accel_mss,speed_ms,0,blend_radius_m)
      movel([0.173673, -1.435888, -2.528156, -0.748344, 1.570796, 1.744469],accel_mss,speed_ms,0,blend_radius_m)
      movel([0.173964, -1.436201, -2.527910, -0.748278, 1.570796, 1.744761],accel_mss,speed_ms,0,blend_radius_m)
      movel([0.174237, -1.436527, -2.527653, -0.748209, 1.570796, 1.745033],accel_mss,speed_ms,0,blend_radius_m)
      movel([0.174499, -1.436860, -2.527390, -0.748139, 1.570796, 1.745295],accel_mss,speed_ms,0,blend_radius_m)
      movel([0.174742, -1.437207, -2.527116, -0.748066, 1.570796, 1.745539],accel_mss,speed_ms,0,blend_radius_m)
      movel([0.174973, -1.437564, -2.526834, -0.747991, 1.570796, 1.745769],accel_mss,speed_ms,0,blend_radius_m)
      movel([0.175187, -1.437932, -2.526543, -0.747914, 1.570796, 1.745983],accel_mss,speed_ms,0,blend_radius_m)
      movel([0.175386, -1.438308, -2.526245, -0.747836, 1.570796, 1.746182],accel_mss,speed_ms,0,blend_radius_m)
      movel([0.175570, -1.438693, -2.525940, -0.747756, 1.570796, 1.746366],accel_mss,speed_ms,0,blend_radius_m)
      movel([0.175738, -1.439089, -2.525626, -0.747674, 1.570796, 1.746535],accel_mss,speed_ms,0,blend_radius_m)
      movel([0.175892, -1.439493, -2.525306, -0.747590, 1.570796, 1.746688],accel_mss,speed_ms,0,blend_radius_m)
      movel([0.176027, -1.439906, -2.524978, -0.747505, 1.570796, 1.746824],accel_mss,speed_ms,0,blend_radius_m)
      movel([0.176148, -1.440326, -2.524645, -0.747419, 1.570796, 1.746944],accel_mss,speed_ms,0,blend_radius_m)
      movel([0.176253, -1.440756, -2.524303, -0.747330, 1.570796, 1.747050],accel_mss,speed_ms,0,blend_radius_m)
      movel([0.176352, -1.441242, -2.523916, -0.747231, 1.570796, 1.747148],accel_mss,speed_ms,0,blend_radius_m)
      movel([0.176433, -1.441734, -2.523524, -0.747131, 1.570796, 1.747230],accel_mss,speed_ms,0,blend_radius_m)
      movel([0.176495, -1.442236, -2.523124, -0.747029, 1.570796, 1.747291],accel_mss,speed_ms,0,blend_radius_m)
      movel([0.176540, -1.442742, -2.522720, -0.746927, 1.570796, 1.747337],accel_mss,speed_ms,0,blend_radius_m)
      movel([0.176568, -1.443257, -2.522308, -0.746824, 1.570796, 1.747364],accel_mss,speed_ms,0,blend_radius_m)
      movel([0.176577, -1.443777, -2.521892, -0.746719, 1.570796, 1.747374],accel_mss,speed_ms,0,blend_radius_m)
      movel([0.176568, -1.444303, -2.521472, -0.746615, 1.570796, 1.747364],accel_mss,speed_ms,0,blend_radius_m)
      movel([0.176541, -1.444834, -2.521046, -0.746509, 1.570796, 1.747338],accel_mss,speed_ms,0,blend_radius_m)
      movel([0.176497, -1.445369, -2.520617, -0.746403, 1.570796, 1.747293],accel_mss,speed_ms,0,blend_radius_m)
      movel([0.176434, -1.445909, -2.520184, -0.746297, 1.570796, 1.747230],accel_mss,speed_ms,0,blend_radius_m)
      movel([0.176354, -1.446453, -2.519746, -0.746190, 1.570796, 1.747150],accel_mss,speed_ms,0,blend_radius_m)
      movel([0.176257, -1.447000, -2.519306, -0.746083, 1.570796, 1.747053],accel_mss,speed_ms,0,blend_radius_m)
      movel([0.176177, -1.447392, -2.518991, -0.746007, 1.570796, 1.746974],accel_mss,speed_ms,0,blend_radius_m)
      movel([0.176085, -1.447785, -2.518674, -0.745930, 1.570796, 1.746881],accel_mss,speed_ms,0,blend_radius_m)
      movel([0.175973, -1.448230, -2.518315, -0.745844, 1.570796, 1.746769],accel_mss,speed_ms,0,blend_radius_m)
      movel([0.175852, -1.448674, -2.517957, -0.745758, 1.570796, 1.746649],accel_mss,speed_ms,0,blend_radius_m)
      movel([0.175731, -1.449101, -2.517612, -0.745676, 1.570796, 1.746528],accel_mss,speed_ms,0,blend_radius_m)
      movel([0.175599, -1.449527, -2.517267, -0.745595, 1.570796, 1.746396],accel_mss,speed_ms,0,blend_radius_m)
      movel([0.175490, -1.449861, -2.516997, -0.745531, 1.570796, 1.746287],accel_mss,speed_ms,0,blend_radius_m)
      movel([0.175366, -1.450195, -2.516726, -0.745467, 1.570796, 1.746162],accel_mss,speed_ms,0,blend_radius_m)
      movel([0.175154, -1.450726, -2.516296, -0.745367, 1.570796, 1.745951],accel_mss,speed_ms,0,blend_radius_m)
      movel([0.174927, -1.451258, -2.515865, -0.745266, 1.570796, 1.745724],accel_mss,speed_ms,0,blend_radius_m)
      movel([0.174685, -1.451788, -2.515435, -0.745166, 1.570796, 1.745482],accel_mss,speed_ms,0,blend_radius_m)
      movel([0.174431, -1.452318, -2.515004, -0.745067, 1.570796, 1.745227],accel_mss,speed_ms,0,blend_radius_m)
      movel([0.174162, -1.452844, -2.514576, -0.744969, 1.570796, 1.744958],accel_mss,speed_ms,0,blend_radius_m)
      movel([0.173880, -1.453371, -2.514147, -0.744871, 1.570796, 1.744676],accel_mss,speed_ms,0,blend_radius_m)
      movel([0.173583, -1.453894, -2.513721, -0.744774, 1.570796, 1.744380],accel_mss,speed_ms,0,blend_radius_m)
      movel([0.173275, -1.454415, -2.513295, -0.744678, 1.570796, 1.744071],accel_mss,speed_ms,0,blend_radius_m)
      movel([0.172952, -1.454933, -2.512872, -0.744583, 1.570796, 1.743748],accel_mss,speed_ms,0,blend_radius_m)
      movel([0.172616, -1.455449, -2.512450, -0.744489, 1.570796, 1.743413],accel_mss,speed_ms,0,blend_radius_m)
      movel([0.172267, -1.455960, -2.512032, -0.744396, 1.570796, 1.743064],accel_mss,speed_ms,0,blend_radius_m)
      movel([0.171921, -1.456447, -2.511634, -0.744308, 1.570796, 1.742717],accel_mss,speed_ms,0,blend_radius_m)
      movel([0.171563, -1.456928, -2.511239, -0.744222, 1.570796, 1.742359],accel_mss,speed_ms,0,blend_radius_m)
      movel([0.171191, -1.457406, -2.510847, -0.744136, 1.570796, 1.741987],accel_mss,speed_ms,0,blend_radius_m)
      movel([0.170805, -1.457879, -2.510459, -0.744051, 1.570796, 1.741601],accel_mss,speed_ms,0,blend_radius_m)
      movel([0.170410, -1.458343, -2.510077, -0.743969, 1.570796, 1.741206],accel_mss,speed_ms,0,blend_radius_m)
      movel([0.170001, -1.458805, -2.509697, -0.743887, 1.570796, 1.740797],accel_mss,speed_ms,0,blend_radius_m)
      movel([0.169581, -1.459256, -2.509325, -0.743807, 1.570796, 1.740377],accel_mss,speed_ms,0,blend_radius_m)
      movel([0.169149, -1.459705, -2.508956, -0.743728, 1.570796, 1.739945],accel_mss,speed_ms,0,blend_radius_m)
      movel([0.168708, -1.460143, -2.508595, -0.743651, 1.570796, 1.739505],accel_mss,speed_ms,0,blend_radius_m)
      movel([0.168257, -1.460573, -2.508240, -0.743576, 1.570796, 1.739053],accel_mss,speed_ms,0,blend_radius_m)
      movel([0.167796, -1.460996, -2.507890, -0.743503, 1.570796, 1.738593],accel_mss,speed_ms,0,blend_radius_m)
      movel([0.167337, -1.461401, -2.507555, -0.743433, 1.570796, 1.738134],accel_mss,speed_ms,0,blend_radius_m)
      movel([0.166868, -1.461797, -2.507228, -0.743364, 1.570796, 1.737664],accel_mss,speed_ms,0,blend_radius_m)
      movel([0.166392, -1.462182, -2.506909, -0.743298, 1.570796, 1.737188],accel_mss,speed_ms,0,blend_radius_m)
      movel([0.165907, -1.462560, -2.506596, -0.743233, 1.570796, 1.736703],accel_mss,speed_ms,0,blend_radius_m)
      movel([0.165413, -1.462928, -2.506291, -0.743170, 1.570796, 1.736209],accel_mss,speed_ms,0,blend_radius_m)
      movel([0.164913, -1.463284, -2.505995, -0.743110, 1.570796, 1.735710],accel_mss,speed_ms,0,blend_radius_m)
      movel([0.164407, -1.463630, -2.505708, -0.743051, 1.570796, 1.735204],accel_mss,speed_ms,0,blend_radius_m)
      movel([0.163895, -1.463965, -2.505430, -0.742994, 1.570796, 1.734691],accel_mss,speed_ms,0,blend_radius_m)
      movel([0.163376, -1.464291, -2.505159, -0.742939, 1.570796, 1.734172],accel_mss,speed_ms,0,blend_radius_m)
      movel([0.162851, -1.464602, -2.504900, -0.742887, 1.570796, 1.733648],accel_mss,speed_ms,0,blend_radius_m)
      movel([0.162323, -1.464904, -2.504649, -0.742836, 1.570796, 1.733119],accel_mss,speed_ms,0,blend_radius_m)
      movel([0.161787, -1.465195, -2.504407, -0.742788, 1.570796, 1.732584],accel_mss,speed_ms,0,blend_radius_m)
      movel([0.161246, -1.465474, -2.504174, -0.742741, 1.570796, 1.732042],accel_mss,speed_ms,0,blend_radius_m)
      movel([0.160703, -1.465741, -2.503952, -0.742697, 1.570796, 1.731499],accel_mss,speed_ms,0,blend_radius_m)
      movel([0.160158, -1.465995, -2.503740, -0.742654, 1.570796, 1.730955],accel_mss,speed_ms,0,blend_radius_m)
      movel([0.159610, -1.466236, -2.503538, -0.742614, 1.570796, 1.730406],accel_mss,speed_ms,0,blend_radius_m)
      movel([0.159059, -1.466465, -2.503347, -0.742576, 1.570796, 1.729855],accel_mss,speed_ms,0,blend_radius_m)
      movel([0.158507, -1.466680, -2.503168, -0.742541, 1.570796, 1.729303],accel_mss,speed_ms,0,blend_radius_m)
      movel([0.157955, -1.466883, -2.502998, -0.742508, 1.570796, 1.728752],accel_mss,speed_ms,0,blend_radius_m)
      movel([0.157402, -1.467072, -2.502840, -0.742477, 1.570796, 1.728198],accel_mss,speed_ms,0,blend_radius_m)
      movel([0.156847, -1.467246, -2.502695, -0.742448, 1.570796, 1.727644],accel_mss,speed_ms,0,blend_radius_m)
      movel([0.156295, -1.467409, -2.502559, -0.742421, 1.570796, 1.727091],accel_mss,speed_ms,0,blend_radius_m)
      movel([0.155666, -1.467577, -2.502418, -0.742394, 1.570796, 1.726462],accel_mss,speed_ms,0,blend_radius_m)
      movel([0.155388, -1.467648, -2.502359, -0.742382, 1.570796, 1.726185],accel_mss,speed_ms,0,blend_radius_m)
      movel([0.155114, -1.467712, -2.502305, -0.742372, 1.570796, 1.725911],accel_mss,speed_ms,0,blend_radius_m)
      movel([0.154653, -1.467815, -2.502219, -0.742355, 1.570796, 1.725449],accel_mss,speed_ms,0,blend_radius_m)
      movel([0.154596, -1.467821, -2.502214, -0.742354, 1.570796, 1.725392],accel_mss,speed_ms,0,blend_radius_m)
      movel([0.154544, -1.467810, -2.502223, -0.742356, 1.570796, 1.725340],accel_mss,speed_ms,0,blend_radius_m)
      movel([0.154517, -1.467791, -2.502239, -0.742359, 1.570796, 1.725313],accel_mss,speed_ms,0,blend_radius_m)
      movel([0.154501, -1.467762, -2.502263, -0.742364, 1.570796, 1.725297],accel_mss,speed_ms,0,blend_radius_m)
      movel([0.154500, -1.467727, -2.502293, -0.742369, 1.570796, 1.725297],accel_mss,speed_ms,0,blend_radius_m)
      movel([0.155344, -1.462784, -2.506410, -0.743195, 1.570796, 1.726141],accel_mss,speed_ms,0,blend_radius_m)
      movel([0.155822, -1.460023, -2.508694, -0.743672, 1.570796, 1.726618],accel_mss,speed_ms,0,blend_radius_m)
      movel([0.156310, -1.457250, -2.510975, -0.744164, 1.570796, 1.727106],accel_mss,speed_ms,0,blend_radius_m)
      movel([0.156901, -1.453946, -2.513678, -0.744765, 1.570796, 1.727698],accel_mss,speed_ms,0,blend_radius_m)
      movel([0.157500, -1.450626, -2.516378, -0.745386, 1.570796, 1.728296],accel_mss,speed_ms,0,blend_radius_m)
      movel([0.160721, -1.433060, -2.530380, -0.748950, 1.570796, 1.731517],accel_mss,speed_ms,0,blend_radius_m)
      movel([0.162422, -1.432812, -2.530574, -0.749003, 1.570796, 1.733218],accel_mss,speed_ms,0,blend_radius_m)
      movel([0.162956, -1.432741, -2.530629, -0.749019, 1.570796, 1.733752],accel_mss,speed_ms,0,blend_radius_m)
      movel([0.163483, -1.432686, -2.530672, -0.749031, 1.570796, 1.734279],accel_mss,speed_ms,0,blend_radius_m)
      movel([0.164006, -1.432647, -2.530703, -0.749039, 1.570796, 1.734803],accel_mss,speed_ms,0,blend_radius_m)
      movel([0.164523, -1.432624, -2.530721, -0.749044, 1.570796, 1.735319],accel_mss,speed_ms,0,blend_radius_m)
      movel([0.165034, -1.432615, -2.530728, -0.749046, 1.570796, 1.735830],accel_mss,speed_ms,0,blend_radius_m)
      movel([0.165538, -1.432623, -2.530722, -0.749044, 1.570796, 1.736334],accel_mss,speed_ms,0,blend_radius_m)
      movel([0.166036, -1.432647, -2.530703, -0.749039, 1.570796, 1.736832],accel_mss,speed_ms,0,blend_radius_m)
      movel([0.166525, -1.432685, -2.530673, -0.749031, 1.570796, 1.737321],accel_mss,speed_ms,0,blend_radius_m)
      movel([0.167009, -1.432738, -2.530632, -0.749019, 1.570796, 1.737805],accel_mss,speed_ms,0,blend_radius_m)
      movel([0.167480, -1.432808, -2.530577, -0.749004, 1.570796, 1.738276],accel_mss,speed_ms,0,blend_radius_m)
      movel([0.167944, -1.432893, -2.530511, -0.748986, 1.570796, 1.738740],accel_mss,speed_ms,0,blend_radius_m)
      movel([0.168398, -1.432991, -2.530433, -0.748965, 1.570796, 1.739194],accel_mss,speed_ms,0,blend_radius_m)
      movel([0.168842, -1.433106, -2.530343, -0.748940, 1.570796, 1.739639],accel_mss,speed_ms,0,blend_radius_m)
      speed_ms = 0.003
      movel([0.168842, -1.436241, -2.531746, -0.744403, 1.570796, 1.739639],accel_mss,speed_ms,0,blend_radius_m)
      speed_ms = 0.007
      movel([0.169285, -1.436373, -2.531641, -0.744375, 1.570796, 1.740082],accel_mss,speed_ms,0,blend_radius_m)
      movel([0.169716, -1.436520, -2.531526, -0.744344, 1.570796, 1.740513],accel_mss,speed_ms,0,blend_radius_m)
      movel([0.170138, -1.436678, -2.531401, -0.744310, 1.570796, 1.740935],accel_mss,speed_ms,0,blend_radius_m)
      movel([0.170548, -1.436853, -2.531263, -0.744273, 1.570796, 1.741344],accel_mss,speed_ms,0,blend_radius_m)
      movel([0.170948, -1.437041, -2.531114, -0.744233, 1.570796, 1.741744],accel_mss,speed_ms,0,blend_radius_m)
      movel([0.171334, -1.437242, -2.530956, -0.744191, 1.570796, 1.742130],accel_mss,speed_ms,0,blend_radius_m)
      movel([0.171708, -1.437458, -2.530786, -0.744145, 1.570796, 1.742505],accel_mss,speed_ms,0,blend_radius_m)
      movel([0.172069, -1.437685, -2.530606, -0.744098, 1.570796, 1.742865],accel_mss,speed_ms,0,blend_radius_m)
      movel([0.172417, -1.437925, -2.530417, -0.744047, 1.570796, 1.743214],accel_mss,speed_ms,0,blend_radius_m)
      movel([0.172752, -1.438179, -2.530216, -0.743994, 1.570796, 1.743548],accel_mss,speed_ms,0,blend_radius_m)
      movel([0.173073, -1.438446, -2.530005, -0.743938, 1.570796, 1.743869],accel_mss,speed_ms,0,blend_radius_m)
      movel([0.173380, -1.438723, -2.529785, -0.743880, 1.570796, 1.744176],accel_mss,speed_ms,0,blend_radius_m)
      movel([0.173673, -1.439015, -2.529554, -0.743820, 1.570796, 1.744469],accel_mss,speed_ms,0,blend_radius_m)
      movel([0.173964, -1.439327, -2.529308, -0.743755, 1.570796, 1.744761],accel_mss,speed_ms,0,blend_radius_m)
      movel([0.174237, -1.439651, -2.529050, -0.743687, 1.570796, 1.745033],accel_mss,speed_ms,0,blend_radius_m)
      movel([0.174499, -1.439984, -2.528786, -0.743619, 1.570796, 1.745295],accel_mss,speed_ms,0,blend_radius_m)
      movel([0.174742, -1.440330, -2.528512, -0.743547, 1.570796, 1.745539],accel_mss,speed_ms,0,blend_radius_m)
      movel([0.174973, -1.440686, -2.528229, -0.743474, 1.570796, 1.745769],accel_mss,speed_ms,0,blend_radius_m)
      movel([0.175187, -1.441053, -2.527938, -0.743399, 1.570796, 1.745983],accel_mss,speed_ms,0,blend_radius_m)
      movel([0.175386, -1.441428, -2.527639, -0.743322, 1.570796, 1.746182],accel_mss,speed_ms,0,blend_radius_m)
      movel([0.175570, -1.441812, -2.527334, -0.743244, 1.570796, 1.746366],accel_mss,speed_ms,0,blend_radius_m)
      movel([0.175738, -1.442206, -2.527019, -0.743163, 1.570796, 1.746535],accel_mss,speed_ms,0,blend_radius_m)
      movel([0.175892, -1.442609, -2.526698, -0.743082, 1.570796, 1.746688],accel_mss,speed_ms,0,blend_radius_m)
      movel([0.176027, -1.443021, -2.526370, -0.742998, 1.570796, 1.746824],accel_mss,speed_ms,0,blend_radius_m)
      movel([0.176148, -1.443440, -2.526036, -0.742914, 1.570796, 1.746944],accel_mss,speed_ms,0,blend_radius_m)
      movel([0.176253, -1.443868, -2.525693, -0.742828, 1.570796, 1.747050],accel_mss,speed_ms,0,blend_radius_m)
      movel([0.176352, -1.444353, -2.525306, -0.742731, 1.570796, 1.747148],accel_mss,speed_ms,0,blend_radius_m)
      movel([0.176433, -1.444844, -2.524913, -0.742633, 1.570796, 1.747230],accel_mss,speed_ms,0,blend_radius_m)
      movel([0.176495, -1.445344, -2.524512, -0.742533, 1.570796, 1.747291],accel_mss,speed_ms,0,blend_radius_m)
      movel([0.176540, -1.445849, -2.524107, -0.742433, 1.570796, 1.747337],accel_mss,speed_ms,0,blend_radius_m)
      movel([0.176568, -1.446362, -2.523695, -0.742332, 1.570796, 1.747364],accel_mss,speed_ms,0,blend_radius_m)
      movel([0.176577, -1.446881, -2.523278, -0.742230, 1.570796, 1.747374],accel_mss,speed_ms,0,blend_radius_m)
      movel([0.176568, -1.447405, -2.522857, -0.742128, 1.570796, 1.747364],accel_mss,speed_ms,0,blend_radius_m)
      movel([0.176541, -1.447935, -2.522430, -0.742024, 1.570796, 1.747338],accel_mss,speed_ms,0,blend_radius_m)
      movel([0.176497, -1.448468, -2.522000, -0.741921, 1.570796, 1.747293],accel_mss,speed_ms,0,blend_radius_m)
      movel([0.176434, -1.449006, -2.521566, -0.741817, 1.570796, 1.747230],accel_mss,speed_ms,0,blend_radius_m)
      movel([0.176354, -1.449549, -2.521128, -0.741712, 1.570796, 1.747150],accel_mss,speed_ms,0,blend_radius_m)
      movel([0.176257, -1.450095, -2.520686, -0.741608, 1.570796, 1.747053],accel_mss,speed_ms,0,blend_radius_m)
      movel([0.176177, -1.450485, -2.520371, -0.741533, 1.570796, 1.746974],accel_mss,speed_ms,0,blend_radius_m)
      movel([0.176085, -1.450877, -2.520053, -0.741459, 1.570796, 1.746881],accel_mss,speed_ms,0,blend_radius_m)
      movel([0.175973, -1.451320, -2.519694, -0.741375, 1.570796, 1.746769],accel_mss,speed_ms,0,blend_radius_m)
      movel([0.175852, -1.451763, -2.519335, -0.741291, 1.570796, 1.746649],accel_mss,speed_ms,0,blend_radius_m)
      movel([0.175731, -1.452189, -2.518989, -0.741211, 1.570796, 1.746528],accel_mss,speed_ms,0,blend_radius_m)
      movel([0.175599, -1.452614, -2.518644, -0.741131, 1.570796, 1.746396],accel_mss,speed_ms,0,blend_radius_m)
      movel([0.175490, -1.452947, -2.518373, -0.741069, 1.570796, 1.746287],accel_mss,speed_ms,0,blend_radius_m)
      movel([0.175366, -1.453280, -2.518102, -0.741007, 1.570796, 1.746162],accel_mss,speed_ms,0,blend_radius_m)
      movel([0.175154, -1.453809, -2.517671, -0.740908, 1.570796, 1.745951],accel_mss,speed_ms,0,blend_radius_m)
      movel([0.174927, -1.454339, -2.517239, -0.740810, 1.570796, 1.745724],accel_mss,speed_ms,0,blend_radius_m)
      movel([0.174685, -1.454868, -2.516808, -0.740713, 1.570796, 1.745482],accel_mss,speed_ms,0,blend_radius_m)
      movel([0.174431, -1.455396, -2.516377, -0.740616, 1.570796, 1.745227],accel_mss,speed_ms,0,blend_radius_m)
      movel([0.174162, -1.455921, -2.515947, -0.740520, 1.570796, 1.744958],accel_mss,speed_ms,0,blend_radius_m)
      movel([0.173880, -1.456446, -2.515518, -0.740425, 1.570796, 1.744676],accel_mss,speed_ms,0,blend_radius_m)
      movel([0.173583, -1.456968, -2.515091, -0.740331, 1.570796, 1.744380],accel_mss,speed_ms,0,blend_radius_m)
      movel([0.173275, -1.457488, -2.514664, -0.740237, 1.570796, 1.744071],accel_mss,speed_ms,0,blend_radius_m)
      movel([0.172952, -1.458004, -2.514241, -0.740144, 1.570796, 1.743748],accel_mss,speed_ms,0,blend_radius_m)
      movel([0.172616, -1.458519, -2.513818, -0.740052, 1.570796, 1.743413],accel_mss,speed_ms,0,blend_radius_m)
      movel([0.172267, -1.459028, -2.513399, -0.739962, 1.570796, 1.743064],accel_mss,speed_ms,0,blend_radius_m)
      movel([0.171921, -1.459513, -2.513000, -0.739876, 1.570796, 1.742717],accel_mss,speed_ms,0,blend_radius_m)
      movel([0.171563, -1.459993, -2.512604, -0.739791, 1.570796, 1.742359],accel_mss,speed_ms,0,blend_radius_m)
      movel([0.171191, -1.460470, -2.512211, -0.739708, 1.570796, 1.741987],accel_mss,speed_ms,0,blend_radius_m)
      movel([0.170805, -1.460941, -2.511823, -0.739625, 1.570796, 1.741601],accel_mss,speed_ms,0,blend_radius_m)
      movel([0.170410, -1.461404, -2.511440, -0.739545, 1.570796, 1.741206],accel_mss,speed_ms,0,blend_radius_m)
      movel([0.170001, -1.461864, -2.511060, -0.739465, 1.570796, 1.740797],accel_mss,speed_ms,0,blend_radius_m)
      movel([0.169581, -1.462315, -2.510687, -0.739387, 1.570796, 1.740377],accel_mss,speed_ms,0,blend_radius_m)
      movel([0.169149, -1.462761, -2.510317, -0.739310, 1.570796, 1.739945],accel_mss,speed_ms,0,blend_radius_m)
      movel([0.168708, -1.463198, -2.509955, -0.739236, 1.570796, 1.739505],accel_mss,speed_ms,0,blend_radius_m)
      movel([0.168257, -1.463627, -2.509599, -0.739162, 1.570796, 1.739053],accel_mss,speed_ms,0,blend_radius_m)
      movel([0.167796, -1.464049, -2.509249, -0.739091, 1.570796, 1.738593],accel_mss,speed_ms,0,blend_radius_m)
      movel([0.167337, -1.464453, -2.508914, -0.739022, 1.570796, 1.738134],accel_mss,speed_ms,0,blend_radius_m)
      movel([0.166868, -1.464847, -2.508586, -0.738956, 1.570796, 1.737664],accel_mss,speed_ms,0,blend_radius_m)
      movel([0.166392, -1.465232, -2.508266, -0.738891, 1.570796, 1.737188],accel_mss,speed_ms,0,blend_radius_m)
      movel([0.165907, -1.465608, -2.507952, -0.738828, 1.570796, 1.736703],accel_mss,speed_ms,0,blend_radius_m)
      movel([0.165413, -1.465975, -2.507647, -0.738767, 1.570796, 1.736209],accel_mss,speed_ms,0,blend_radius_m)
      movel([0.164913, -1.466330, -2.507351, -0.738708, 1.570796, 1.735710],accel_mss,speed_ms,0,blend_radius_m)
      movel([0.164407, -1.466675, -2.507063, -0.738651, 1.570796, 1.735204],accel_mss,speed_ms,0,blend_radius_m)
      movel([0.163895, -1.467009, -2.506784, -0.738596, 1.570796, 1.734691],accel_mss,speed_ms,0,blend_radius_m)
      movel([0.163376, -1.467334, -2.506513, -0.738542, 1.570796, 1.734172],accel_mss,speed_ms,0,blend_radius_m)
      movel([0.162851, -1.467645, -2.506253, -0.738491, 1.570796, 1.733648],accel_mss,speed_ms,0,blend_radius_m)
      movel([0.162323, -1.467945, -2.506002, -0.738442, 1.570796, 1.733119],accel_mss,speed_ms,0,blend_radius_m)
      movel([0.161787, -1.468235, -2.505759, -0.738394, 1.570796, 1.732584],accel_mss,speed_ms,0,blend_radius_m)
      movel([0.161246, -1.468514, -2.505526, -0.738349, 1.570796, 1.732042],accel_mss,speed_ms,0,blend_radius_m)
      movel([0.160703, -1.468780, -2.505303, -0.738306, 1.570796, 1.731499],accel_mss,speed_ms,0,blend_radius_m)
      movel([0.160158, -1.469033, -2.505091, -0.738265, 1.570796, 1.730955],accel_mss,speed_ms,0,blend_radius_m)
      movel([0.159610, -1.469274, -2.504889, -0.738226, 1.570796, 1.730406],accel_mss,speed_ms,0,blend_radius_m)
      movel([0.159059, -1.469502, -2.504698, -0.738189, 1.570796, 1.729855],accel_mss,speed_ms,0,blend_radius_m)
      movel([0.158507, -1.469716, -2.504518, -0.738155, 1.570796, 1.729303],accel_mss,speed_ms,0,blend_radius_m)
      movel([0.157955, -1.469919, -2.504348, -0.738122, 1.570796, 1.728752],accel_mss,speed_ms,0,blend_radius_m)
      movel([0.157402, -1.470107, -2.504190, -0.738092, 1.570796, 1.728198],accel_mss,speed_ms,0,blend_radius_m)
      movel([0.156847, -1.470281, -2.504044, -0.738064, 1.570796, 1.727644],accel_mss,speed_ms,0,blend_radius_m)
      movel([0.156295, -1.470443, -2.503908, -0.738038, 1.570796, 1.727091],accel_mss,speed_ms,0,blend_radius_m)
      movel([0.155666, -1.470611, -2.503767, -0.738011, 1.570796, 1.726462],accel_mss,speed_ms,0,blend_radius_m)
      movel([0.155388, -1.470681, -2.503708, -0.738000, 1.570796, 1.726185],accel_mss,speed_ms,0,blend_radius_m)
      movel([0.155114, -1.470745, -2.503654, -0.737990, 1.570796, 1.725911],accel_mss,speed_ms,0,blend_radius_m)
      movel([0.154653, -1.470848, -2.503568, -0.737974, 1.570796, 1.725449],accel_mss,speed_ms,0,blend_radius_m)
      movel([0.154596, -1.470853, -2.503563, -0.737973, 1.570796, 1.725392],accel_mss,speed_ms,0,blend_radius_m)
      movel([0.154544, -1.470843, -2.503572, -0.737974, 1.570796, 1.725340],accel_mss,speed_ms,0,blend_radius_m)
      movel([0.154517, -1.470824, -2.503588, -0.737978, 1.570796, 1.725313],accel_mss,speed_ms,0,blend_radius_m)
      movel([0.154501, -1.470795, -2.503612, -0.737982, 1.570796, 1.725297],accel_mss,speed_ms,0,blend_radius_m)
      movel([0.154500, -1.470760, -2.503642, -0.737988, 1.570796, 1.725297],accel_mss,speed_ms,0,blend_radius_m)
      movel([0.155344, -1.465832, -2.507766, -0.738791, 1.570796, 1.726141],accel_mss,speed_ms,0,blend_radius_m)
      movel([0.155822, -1.463079, -2.510054, -0.739256, 1.570796, 1.726618],accel_mss,speed_ms,0,blend_radius_m)
      movel([0.156310, -1.460314, -2.512340, -0.739735, 1.570796, 1.727106],accel_mss,speed_ms,0,blend_radius_m)
      movel([0.156901, -1.457020, -2.515048, -0.740321, 1.570796, 1.727698],accel_mss,speed_ms,0,blend_radius_m)
      movel([0.157500, -1.453709, -2.517753, -0.740927, 1.570796, 1.728296],accel_mss,speed_ms,0,blend_radius_m)
      movel([0.160721, -1.436194, -2.531782, -0.744413, 1.570796, 1.731517],accel_mss,speed_ms,0,blend_radius_m)
      movel([0.162422, -1.435948, -2.531976, -0.744465, 1.570796, 1.733218],accel_mss,speed_ms,0,blend_radius_m)
      movel([0.162956, -1.435877, -2.532032, -0.744480, 1.570796, 1.733752],accel_mss,speed_ms,0,blend_radius_m)
      movel([0.163483, -1.435822, -2.532075, -0.744492, 1.570796, 1.734279],accel_mss,speed_ms,0,blend_radius_m)
      movel([0.164006, -1.435783, -2.532106, -0.744500, 1.570796, 1.734803],accel_mss,speed_ms,0,blend_radius_m)
      movel([0.164523, -1.435760, -2.532124, -0.744505, 1.570796, 1.735319],accel_mss,speed_ms,0,blend_radius_m)
      movel([0.165034, -1.435752, -2.532131, -0.744507, 1.570796, 1.735830],accel_mss,speed_ms,0,blend_radius_m)
      movel([0.165538, -1.435759, -2.532125, -0.744505, 1.570796, 1.736334],accel_mss,speed_ms,0,blend_radius_m)
      movel([0.166036, -1.435783, -2.532106, -0.744500, 1.570796, 1.736832],accel_mss,speed_ms,0,blend_radius_m)
      movel([0.166525, -1.435821, -2.532076, -0.744492, 1.570796, 1.737321],accel_mss,speed_ms,0,blend_radius_m)
      movel([0.167009, -1.435874, -2.532035, -0.744481, 1.570796, 1.737805],accel_mss,speed_ms,0,blend_radius_m)
      movel([0.167480, -1.435943, -2.531980, -0.744466, 1.570796, 1.738276],accel_mss,speed_ms,0,blend_radius_m)
      movel([0.167944, -1.436028, -2.531913, -0.744448, 1.570796, 1.738740],accel_mss,speed_ms,0,blend_radius_m)
      movel([0.168398, -1.436126, -2.531836, -0.744427, 1.570796, 1.739194],accel_mss,speed_ms,0,blend_radius_m)
      movel([0.168842, -1.436241, -2.531746, -0.744403, 1.570796, 1.739639],accel_mss,speed_ms,0,blend_radius_m)
      speed_ms = 0.003
      movel([0.168842, -1.423819, -2.526086, -0.762484, 1.570796, 1.739639],accel_mss,speed_ms,0,blend_radius_m)
      speed_ms = 0.01
      movel([0.168842, -1.399903, -2.514375, -0.798111, 1.570796, 1.739639],accel_mss,speed_ms,0,blend_radius_m)
      movel([0.357278, -1.356224, -2.545602, -0.810563, 1.570796, 1.928074],accel_mss,speed_ms,0,blend_radius_m)
      movel([0.357278, -1.380960, -2.557859, -0.773571, 1.570796, 1.928074],accel_mss,speed_ms,0,blend_radius_m)
      speed_ms = 0.003
      movel([0.357278, -1.390593, -2.562320, -0.759476, 1.570796, 1.928074],accel_mss,speed_ms,0,blend_radius_m)
      speed_ms = 0.007
      movel([0.357356, -1.390308, -2.562525, -0.759556, 1.570796, 1.928153],accel_mss,speed_ms,0,blend_radius_m)
      movel([0.357448, -1.390019, -2.562734, -0.759637, 1.570796, 1.928245],accel_mss,speed_ms,0,blend_radius_m)
      movel([0.357553, -1.389731, -2.562941, -0.759717, 1.570796, 1.928350],accel_mss,speed_ms,0,blend_radius_m)
      movel([0.357672, -1.389442, -2.563149, -0.759798, 1.570796, 1.928469],accel_mss,speed_ms,0,blend_radius_m)
      movel([0.357806, -1.389150, -2.563359, -0.759880, 1.570796, 1.928603],accel_mss,speed_ms,0,blend_radius_m)
      movel([0.357953, -1.388862, -2.563566, -0.759962, 1.570796, 1.928749],accel_mss,speed_ms,0,blend_radius_m)
      movel([0.358142, -1.388509, -2.563819, -0.760061, 1.570796, 1.928938],accel_mss,speed_ms,0,blend_radius_m)
      movel([0.358341, -1.388157, -2.564072, -0.760160, 1.570796, 1.929137],accel_mss,speed_ms,0,blend_radius_m)
      movel([0.358546, -1.387806, -2.564324, -0.760260, 1.570796, 1.929342],accel_mss,speed_ms,0,blend_radius_m)
      movel([0.358793, -1.387411, -2.564607, -0.760372, 1.570796, 1.929589],accel_mss,speed_ms,0,blend_radius_m)
      movel([0.359056, -1.387017, -2.564889, -0.760484, 1.570796, 1.929853],accel_mss,speed_ms,0,blend_radius_m)
      movel([0.359336, -1.386628, -2.565167, -0.760594, 1.570796, 1.930132],accel_mss,speed_ms,0,blend_radius_m)
      movel([0.359627, -1.386244, -2.565442, -0.760704, 1.570796, 1.930424],accel_mss,speed_ms,0,blend_radius_m)
      movel([0.359936, -1.385863, -2.565714, -0.760813, 1.570796, 1.930733],accel_mss,speed_ms,0,blend_radius_m)
      movel([0.360247, -1.385501, -2.565972, -0.760916, 1.570796, 1.931043],accel_mss,speed_ms,0,blend_radius_m)
      movel([0.360574, -1.385145, -2.566226, -0.761018, 1.570796, 1.931370],accel_mss,speed_ms,0,blend_radius_m)
      movel([0.360915, -1.384795, -2.566476, -0.761119, 1.570796, 1.931711],accel_mss,speed_ms,0,blend_radius_m)
      movel([0.361265, -1.384455, -2.566718, -0.761217, 1.570796, 1.932062],accel_mss,speed_ms,0,blend_radius_m)
      movel([0.361629, -1.384123, -2.566954, -0.761312, 1.570796, 1.932425],accel_mss,speed_ms,0,blend_radius_m)
      movel([0.361998, -1.383809, -2.567177, -0.761403, 1.570796, 1.932794],accel_mss,speed_ms,0,blend_radius_m)
      movel([0.362374, -1.383503, -2.567395, -0.761491, 1.570796, 1.933171],accel_mss,speed_ms,0,blend_radius_m)
      movel([0.362763, -1.383210, -2.567603, -0.761576, 1.570796, 1.933559],accel_mss,speed_ms,0,blend_radius_m)
      movel([0.363157, -1.382930, -2.567802, -0.761657, 1.570796, 1.933954],accel_mss,speed_ms,0,blend_radius_m)
      movel([0.363562, -1.382660, -2.567993, -0.761736, 1.570796, 1.934358],accel_mss,speed_ms,0,blend_radius_m)
      movel([0.363972, -1.382406, -2.568173, -0.761810, 1.570796, 1.934768],accel_mss,speed_ms,0,blend_radius_m)
      movel([0.364386, -1.382165, -2.568344, -0.761880, 1.570796, 1.935183],accel_mss,speed_ms,0,blend_radius_m)
      movel([0.364807, -1.381937, -2.568506, -0.761946, 1.570796, 1.935604],accel_mss,speed_ms,0,blend_radius_m)
      movel([0.365231, -1.381726, -2.568655, -0.762008, 1.570796, 1.936027],accel_mss,speed_ms,0,blend_radius_m)
      movel([0.365658, -1.381529, -2.568795, -0.762065, 1.570796, 1.936454],accel_mss,speed_ms,0,blend_radius_m)
      movel([0.366192, -1.381301, -2.568956, -0.762132, 1.570796, 1.936988],accel_mss,speed_ms,0,blend_radius_m)
      movel([0.366727, -1.381083, -2.569110, -0.762196, 1.570796, 1.937523],accel_mss,speed_ms,0,blend_radius_m)
      movel([0.366947, -1.381003, -2.569167, -0.762219, 1.570796, 1.937744],accel_mss,speed_ms,0,blend_radius_m)
